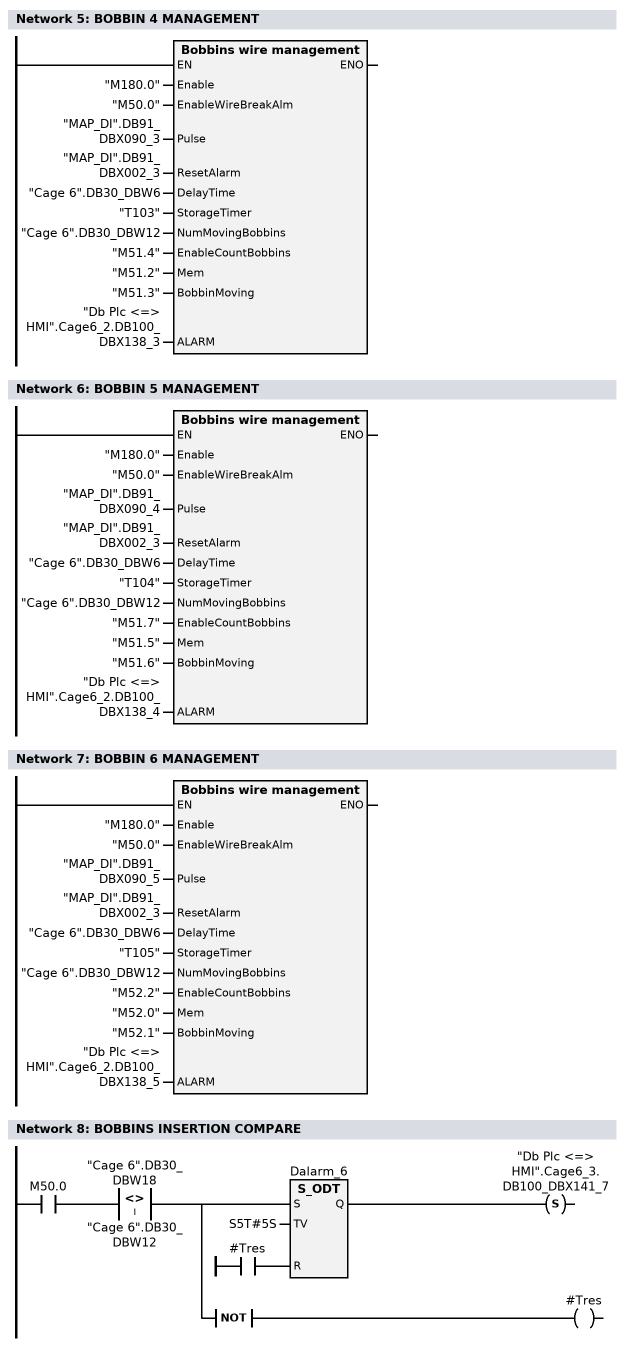
[picture p57: Cage 6 wires insertion networks 5-8]
NETWORK
TITLE = BOBBIN 4 MANAGEMENT
      CALL  "Bobbins wire management" (
           Enable                   := "M180.0",
           EnableWireBreakAlm       := "M50.0",
           Pulse                    := "MAP_DI".DB91_DBX090_3,
           ResetAlarm               := "MAP_DI".DB91_DBX002_3,
           DelayTime                := "Cage 6".DB30_DBW6,
           StorageTimer             := "T103",
           NumMovingBobbins         := "Cage 6".DB30_DBW12,
           EnableCountBobbins       := "M51.4",
           Mem                      := "M51.2",
           BobbinMoving             := "M51.3",
           ALARM                    := "Db Plc <=> HMI".Cage6_2.DB100_DBX138_3);
NETWORK
TITLE = BOBBIN 5 MANAGEMENT
      CALL  "Bobbins wire management" (
           Enable                   := "M180.0",
           EnableWireBreakAlm       := "M50.0",
           Pulse                    := "MAP_DI".DB91_DBX090_4,
           ResetAlarm               := "MAP_DI".DB91_DBX002_3,
           DelayTime                := "Cage 6".DB30_DBW6,
           StorageTimer             := "T104",
           NumMovingBobbins         := "Cage 6".DB30_DBW12,
           EnableCountBobbins       := "M51.7",
           Mem                      := "M51.5",
           BobbinMoving             := "M51.6",
           ALARM                    := "Db Plc <=> HMI".Cage6_2.DB100_DBX138_4);
NETWORK
TITLE = BOBBIN 6 MANAGEMENT
      CALL  "Bobbins wire management" (
           Enable                   := "M180.0",
           EnableWireBreakAlm       := "M50.0",
           Pulse                    := "MAP_DI".DB91_DBX090_5,
           ResetAlarm               := "MAP_DI".DB91_DBX002_3,
           DelayTime                := "Cage 6".DB30_DBW6,
           StorageTimer             := "T105",
           NumMovingBobbins         := "Cage 6".DB30_DBW12,
           EnableCountBobbins       := "M52.2",
           Mem                      := "M52.0",
           BobbinMoving             := "M52.1",
           ALARM                    := "Db Plc <=> HMI".Cage6_2.DB100_DBX138_5);
NETWORK
TITLE = BOBBINS INSERTION COMPARE
      A     "M50.0";
      A(;
      L     "Cage 6".DB30_DBW18;
      L     "Cage 6".DB30_DBW12;
      <>I;
      );
      =     L 1.0;
      A     L 1.0;
      L     S5T#5S;
      SD    "Dalarm_6";
      A     #Tres;
      R     "Dalarm_6";
      NOP   0;
      NOP   0;
      A     "Dalarm_6";
      S     "Db Plc <=> HMI".Cage6_3.DB100_DBX141_7;
      A     L 1.0;
      NOT;
      =     #Tres;
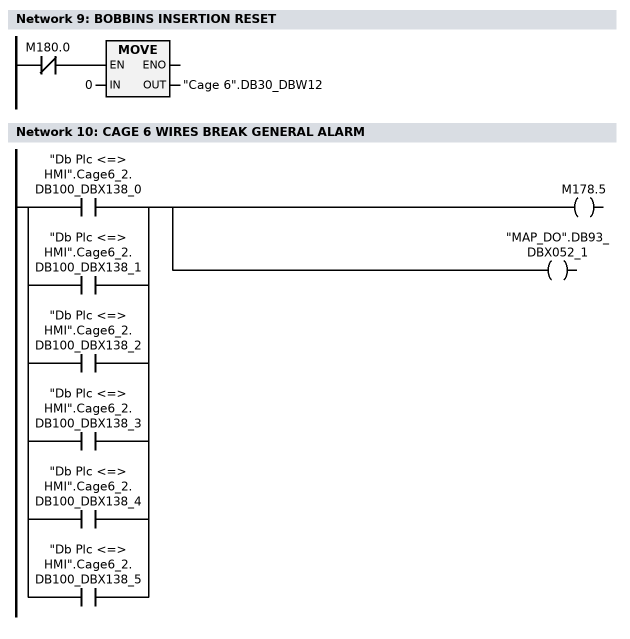
NETWORK
TITLE = BOBBINS INSERTION RESET
      AN    "M180.0";
      JNB   _001;
      L     0;
      T     "Cage 6".DB30_DBW12;
_001: NOP   0;
NETWORK
TITLE = CAGE 6 WIRES BREAK GENERAL ALARM
      O     "Db Plc <=> HMI".Cage6_2.DB100_DBX138_0;
      O     "Db Plc <=> HMI".Cage6_2.DB100_DBX138_1;
      O     "Db Plc <=> HMI".Cage6_2.DB100_DBX138_2;
      O     "Db Plc <=> HMI".Cage6_2.DB100_DBX138_3;
      O     "Db Plc <=> HMI".Cage6_2.DB100_DBX138_4;
      O     "Db Plc <=> HMI".Cage6_2.DB100_DBX138_5;
      =     "M178.5";
      =     "MAP_DO".DB93_DBX052_1;
END_FUNCTION

FUNCTION "Wires break time" : VOID	// FC 74
TITLE = WIRES BREAK TIME FUNCTION
AUTHOR : Milesi
VERSION : 0.1
BEGIN
NETWORK
TITLE = TIME FOR WIRES BREAK CONTROL
//Time for 1 rpm = 60s/Bobbin rpm
//==
//Time for 1 rpm = 60s/(Linear speed/3.141592 * Bobbin Ш)
//==
//Time for 1 rpm = 60/[60000/(3.1415 * 630)] = 1.9792 (s)
//
//In this case for having a good safety margin on the control I do not divide for 
//4 (number fields) but for 3
//
//Time of 1 sector = 1.9792/3 = 0.6597 (s)
//
//Time of 1 sector = K/Linear speed
//==
//K = Linear speed max (mm)*Time of 1 sector (s)/10
//
//K = (60000*0.6597)/10 = 3958.2
//
//Divided 10 for having the time in compatible esadecimale with the base times 
//STEP7 in tenth of second   
      L     3.958200e+03;
      L     "Line".DB55_DBD68;
      /R;
      RND;
      DTB;
      SRW   4;
      L     W#16#1000;
      OW;
      T     "Cage 24".DB15_DBW6;
      T     "Cage 18".DB20_DBW6;
      T     "Cage 12".DB25_DBW6;
      T     "Cage 6".DB30_DBW6;
      T     "Pay-off 630".DB35_DBW6;
END_FUNCTION

FUNCTION "Bobbins diameter" : VOID	// FC 79
TITLE = BOBBINS DIAMETER FUNCTION
AUTHOR : Milesi
VERSION : 0.1
VAR_TEMP
  Enable_24 : BOOL ;
  Enable_18 : BOOL ;
  Enable_12 : BOOL ;
  Enable_6 : BOOL ;
  PayOff_630_Enable : BOOL ;
  PayOff_Enable : BOOL ;
  PayOff_630_Reset : BOOL ;
  PayOff_Reset : BOOL ;
  PayOff_Bobbin_Reset : BOOL ;
END_VAR
BEGIN
NETWORK
TITLE = CAGE 24 DIAMETER CALCULATION
//E47.1 = 4 impulse     
//
      A     "M201.0";
      A     "M192.0";
      =     #Enable_24;
      CALL  "Bobbin diameter calculat" (
           Enable                   := #Enable_24,
           Pulse                    := "MAP_DI".DB91_DBX030_0,
           Pulse_1minute            := "M100.0",
           Reset                    := "M180.7",
           LinearSpeed              := "Line".DB55_DBD68,
           CompattingFactorHMI      := "Cage 24".DB15_DBD28,
           MinDiameterLimit         := 3.550000e+02,
           MaxDiameterLimit         := 6.300000e+02,
           Pulses_number            := 4,
           Mem                      := "M18.4",
           ImpulseForMinRegister    := "Cage 24".DB15_DBW16,
           Diameter                 := "Cage 24".DB15_DBW14);
NETWORK
TITLE = CAGE 18 DIAMETER CALCULATION
//E57.1 = 4 impulse  
      A     "M201.0";
      A     "M186.0";
      =     #Enable_18;
      CALL  "Bobbin diameter calculat" (
           Enable                   := #Enable_18,
           Pulse                    := "MAP_DI".DB91_DBX050_0,
           Pulse_1minute            := "M100.0",
           Reset                    := "M180.6",
           LinearSpeed              := "Line".DB55_DBD68,
           CompattingFactorHMI      := "Cage 18".DB20_DBD28,
           MinDiameterLimit         := 3.550000e+02,
           MaxDiameterLimit         := 6.300000e+02,
           Pulses_number            := 4,
           Mem                      := "M18.3",
           ImpulseForMinRegister    := "Cage 18".DB20_DBW16,
           Diameter                 := "Cage 18".DB20_DBW14);
NETWORK
TITLE = CAGE 12 DIAMETER CALCULATION
//E67.1 = 4 impulse
      A     "M201.0";
      A     "M188.0";
      =     #Enable_12;
      CALL  "Bobbin diameter calculat" (
           Enable                   := #Enable_12,
           Pulse                    := "MAP_DI".DB91_DBX070_0,
           Pulse_1minute            := "M100.0",
           Reset                    := "M180.5",
           LinearSpeed              := "Line".DB55_DBD68,
           CompattingFactorHMI      := "Cage 12".DB25_DBD28,
           MinDiameterLimit         := 3.550000e+02,
           MaxDiameterLimit         := 6.300000e+02,
           Pulses_number            := 4,
           Mem                      := "M18.2",
           ImpulseForMinRegister    := "Cage 12".DB25_DBW16,
           Diameter                 := "Cage 12".DB25_DBW14);
NETWORK
TITLE = CAGE 6 DIAMETER CALCULATION
//E77.1 = 4 impulse 
      A     "M201.0";
      A     "M190.0";
      =     #Enable_6;
      CALL  "Bobbin diameter calculat" (
           Enable                   := #Enable_6,
           Pulse                    := "MAP_DI".DB91_DBX090_0,
           Pulse_1minute            := "M100.0",
           Reset                    := "M180.4",
           LinearSpeed              := "Line".DB55_DBD68,
           CompattingFactorHMI      := 0.000000e+00,
           MinDiameterLimit         := 3.550000e+02,
           MaxDiameterLimit         := 6.300000e+02,
           Pulses_number            := 4,
           Mem                      := "M18.1",
           ImpulseForMinRegister    := "Cage 6".DB30_DBW16,
           Diameter                 := "Cage 6".DB30_DBW14);
NETWORK
TITLE = PAY-OFF 630 DIAMETER CALCULATION
//E79.0 = 4 impulse
      A     "M201.0";
      A     "Pay-off 630".HMI_Bit.DB35_DBX1_7;
      =     #PayOff_630_Enable;
      A     "T0";
      AN    "M180.1";
      AN    "MAP_DI".DB91_DBX099_0;
      =     #PayOff_630_Reset;
      CALL  "Bobbin diameter calculat" (
           Enable                   := #PayOff_630_Enable,
           Pulse                    := "MAP_DI".DB91_DBX099_1,
           Pulse_1minute            := "M100.0",
           Reset                    := #PayOff_630_Reset,
           LinearSpeed              := "Line".DB55_DBD68,
           CompattingFactorHMI      := 0.000000e+00,
           MinDiameterLimit         := 3.550000e+02,
           MaxDiameterLimit         := 6.300000e+02,
           Pulses_number            := 4,
           Mem                      := "M19.0",
           ImpulseForMinRegister    := "Pay-off 630".DB35_DBW16,
           Diameter                 := "Pay-off 630".DB35_DBW14);
NETWORK
TITLE = BOBBINS DIAMETER CALCULATION TIME 
      A     "M201.0";
      AN    "M100.0";
      L     S5T#1M;
      SD    "T5";
      NOP   0;
      NOP   0;
      NOP   0;
      A     "T5";
      =     "M100.0";
END_FUNCTION

FUNCTION "Bobbins brake" : VOID	// FC 80
TITLE = BOBBINS BRAKE OUT FUNCTION
AUTHOR : Milesi
VERSION : 0.1
VAR_TEMP
  Cage12_output : DINT ;
  Cage18_output : DINT ;
  Cage24_output : DINT ;
  pay_of_630_output : DINT ;
  Cage6_output : DINT ;
  pay_bobbin_output : DINT ;
END_VAR
BEGIN
NETWORK
TITLE = CAGE 24 BOBBINS BRAKES OUTPUT
      L     "Cage 24".DB15_DBD128;
      L     "Cage 24".DB15_DBW14;
      ITD;
      DTR;
      *R;
      L     6.300000e+04;
      /R;
      L     2.764800e+04;
      *R;
      RND;
      L     27648;
      >=D;
      JC    OUT1;
      TAK;
OUT1: T     "-659Y2";
NETWORK
TITLE = CAGE 18 BOBBINS BRAKES OUTPUT
      L     "Cage 18".DB20_DBD128;
      L     "Cage 18".DB20_DBW14;
      ITD;
      DTR;
      *R;
      L     6.300000e+04;
      /R;
      L     2.764800e+04;
      *R;
      RND;
      L     27648;
      >=D;
      JC    OUT2;
      TAK;
OUT2: T     "-559Y2";
NETWORK
TITLE = CAGE 12 BOBBINS BRAKES OUTPUT
      L     "Cage 12".DB25_DBD128;
      L     "Cage 12".DB25_DBW14;
      ITD;
      DTR;
      *R;
      L     6.300000e+04;
      /R;
      L     2.764800e+04;
      *R;
      RND;
      L     27648;
      >=D;
      JC    OUT3;
      TAK;
OUT3: T     "PAW288";
NETWORK
TITLE = CAGE 6 BOBBINS BRAKES OUTPUT
      L     "Cage 6".DB30_DBD128;
      L     "Cage 6".DB30_DBW14;
      ITD;
      DTR;
      *R;
      L     6.300000e+04;
      /R;
      L     2.764800e+04;
      *R;
      RND;
      L     27648;
      >=D;
      JC    OUT4;
      TAK;
OUT4: T     "-359Y2";
NETWORK
TITLE = PAY-OFF 630 BOBBIN BRAKE OUTPUT
      L     "Pay-off 630".DB35_DBD20;
      L     "Pay-off 630".DB35_DBW14;
      ITD;
      DTR;
      *R;
      L     6.300000e+04;
      /R;
      L     2.764800e+04;
      *R;
      RND;
      L     27648;
      >=D;
      JC    OUT5;
      TAK;
OUT5: AN    "MAP_DI".DB91_DBX099_4;
      O     "M180.1";
      JC    OUT6;
      L     0;
OUT6: T     "-359Y4";
END_FUNCTION

FUNCTION "Rpm increase" : VOID	// FC 81
TITLE = RPM INCREASE FUNCTION
AUTHOR : Milesi
VERSION : 0.1
VAR_TEMP
  Time_sec : INT ;	//Minuts in seconds
END_VAR
BEGIN
NETWORK
TITLE = STEP TO MAKE 
//Bobbin max Ш - Bobbin min Ш
//630 - 355 = 275
      L     2.750000e+02;
      L     "Line".DB55_DBD156;
      /R;
      T     "Line".DB55_DBD176;
      L     1.000000e+00;
      -R;
      T     "Line".DB55_DBD184;
NETWORK
TITLE = LINEAR SPEED INCREASE FOR SINGLE STEP 
      L     "Line".DB55_DBD40;
      L     "Line".DB55_DBD72;
      -R;
      L     "Line".DB55_DBD184;
      /R;
      T     "Line".DB55_DBD196;
NETWORK
TITLE = LINEAR SPEED INCREASE CONTROL TIME
      A     "M180.1";
      A     "M201.0";
      JNB   OUT;
      A     "M3.5";
      JNB   CLOC;
      L     "Line".DB55_DBD168;
      L     1.000000e+00;
      +R;
      T     "Line".DB55_DBD168;
CLOC: JU    EXIT;
NETWORK
TITLE = LINEAR SPEED INCREASE PARAMETERS RESET
OUT:  L     0.000000e+00;
      T     "Line".DB55_DBD168;
      A     "M180.1";
      JC    EXIT;
      L     6.300000e+02;
      T     "Line".DB55_DBD172;
      L     0.000000e+00;
      T     "Line".DB55_DBD164;
      L     0.000000e+00;
      T     "Line".DB55_DBD76;
EXIT: NOP   0;
NETWORK
TITLE = LINEAR SPEED INCREASE TIME MINUTS TO SECONDS COVERSION
      L     "Line".DB55_DBD160;
      RND;
      T     #Time_sec;
NETWORK
TITLE = DIAMETER NEXT STEP
      L     "Line".DB55_DBD172;
      L     "Line".DB55_DBD156;
      -R;
      T     "Line".DB55_DBD188;
NETWORK
TITLE = LINEAR SPEED INCREASE CONTROL 
      L     "Line".DB55_DBD168;
      RND;
      L     #Time_sec;
      <I;
      BEC;
      L     0.000000e+00;
      T     "Line".DB55_DBD168;
NETWORK
TITLE = LINE LINEAR SPEED INCREASE
      A(;
      L     "Line".DB55_DBD188;
      L     "Line".DB55_DBD192;
      <R;
      );
      O(;
      L     "Line".DB55_DBD164;
      L     "Line".DB55_DBD184;
      >=R;
      );
      BEC;
      L     "Line".DB55_DBD164;
      L     1.000000e+00;
      +R;
      T     "Line".DB55_DBD164;
      L     "Line".DB55_DBD188;
      T     "Line".DB55_DBD172;
      L     "Line".DB55_DBD164;
      L     "Line".DB55_DBD196;
      *R;
      T     "Line".DB55_DBD76;
END_FUNCTION

FUNCTION "Map Input Function" : VOID	// FC 91
TITLE = MAP INPUT FUNCTION
VERSION : 0.1
VAR_TEMP
  Temp1 : BOOL ;
END_VAR
BEGIN
NETWORK
TITLE = da DB91.dbx0.0 a DB91.dbx0.7
      A     "-126K1:Auxiliary";
      =     "MAP_DI".DB91_DBX000_0;
      A     "-126K4";
      =     "MAP_DI".DB91_DBX000_1;
      A     "-175S3";
      =     "MAP_DI".DB91_DBX000_2;
      A     "-112Q3";
      =     "MAP_DI".DB91_DBX000_3;
      A     "-108G1:Alarm";
      =     "MAP_DI".DB91_DBX000_4;
      A     "-108G1:Bat ok";
      =     "MAP_DI".DB91_DBX000_5;
      A     "-116Q1";
      =     "MAP_DI".DB91_DBX000_6;
      CLR;
      =     "MAP_DI".DB91_DBX000_7;
NETWORK
TITLE = da DB91.dbx1.0 a DB91.dbx1.7
      A     "-119Q1";
      =     "MAP_DI".DB91_DBX001_0;
      A     "-141R1:T2";
      =     "MAP_DI".DB91_DBX001_1;
      A     "-140G1:X104:20";
      =     "MAP_DI".DB91_DBX001_2;
      CLR;
      =     "MAP_DI".DB91_DBX001_3;
      =     "MAP_DI".DB91_DBX001_4;
      =     "MAP_DI".DB91_DBX001_5;
      =     "MAP_DI".DB91_DBX001_6;
      =     "MAP_DI".DB91_DBX001_7;
NETWORK
TITLE = da DB91.dbx2.0 a DB91.dbx2.7
      A     "-177S1";
      =     "MAP_DI".DB91_DBX002_0;
      A     "-177S2";
      =     "MAP_DI".DB91_DBX002_1;
      A     "-177S3";
      =     "MAP_DI".DB91_DBX002_2;
      A     "-177S4";
      =     "MAP_DI".DB91_DBX002_3;
      A     "-177S5";
      =     "MAP_DI".DB91_DBX002_4;
      A     "-112K1";
      =     "MAP_DI".DB91_DBX002_5;
      A     "-112K1:66";
      =     "MAP_DI".DB91_DBX002_6;
      A     "-113G1:4";
      =     "MAP_DI".DB91_DBX002_7;
NETWORK
TITLE = da DB91.dbx3.0 a DB91.dbx3.7
      A     "-113G1:3";
      =     "MAP_DI".DB91_DBX003_0;
      A     "-109Q6";
      =     "MAP_DI".DB91_DBX003_1;
      A     "-115Q1";
      =     "MAP_DI".DB91_DBX003_2;
      A     "-140Q1";
      =     "MAP_DI".DB91_DBX003_3;
      A     "-109Q2";
      =     "MAP_DI".DB91_DBX003_4;
      CLR;
      =     "MAP_DI".DB91_DBX003_5;
      =     "MAP_DI".DB91_DBX003_6;
      =     "MAP_DI".DB91_DBX003_7;
NETWORK
TITLE = da DB91.dbx4.0 a DB91.dbx4.7
      A     "-922S5";
      =     "MAP_DI".DB91_DBX004_0;
      A     "-922S6";
      =     "MAP_DI".DB91_DBX004_1;
      A     "-922S7";
      =     "MAP_DI".DB91_DBX004_2;
      A     "-922S8";
      =     "MAP_DI".DB91_DBX004_3;
      A     "-945Q1";
      =     "MAP_DI".DB91_DBX004_4;
      A     "-941Q2";
      =     "MAP_DI".DB91_DBX004_5;
      A     "-964S1:Forward";
      =     "MAP_DI".DB91_DBX004_6;
      A     "-964S1:Backward";
      =     "MAP_DI".DB91_DBX004_7;
NETWORK
TITLE = da DB91.dbx5.0 a DB91.dbx5.7
      L     B#16#0;
      T     DB91.DBB 5;
NETWORK
TITLE = da DB91.dbx6.0 a DB91.dbx6.7
      A     "-961S1";
      =     "MAP_DI".DB91_DBX006_0;
      A     "-961S2";
      =     "MAP_DI".DB91_DBX006_1;
      A     "-961S3";
      =     "MAP_DI".DB91_DBX006_2;
      A     "-961S4";
      =     "MAP_DI".DB91_DBX006_3;
      A     "-961S5:UP";
      =     "MAP_DI".DB91_DBX006_4;
      A     "-961S5:DOWN";
      =     "MAP_DI".DB91_DBX006_5;
      A     "-961S7:UP";
      =     "MAP_DI".DB91_DBX006_6;
      A     "-961S7:DOWN";
      =     "MAP_DI".DB91_DBX006_7;
NETWORK
TITLE = da DB91.dbx7.0 a DB91.dbx7.7
      A     "-962S1:UP";
      =     "MAP_DI".DB91_DBX007_0;
      A     "-962S1:DOWN";
      =     "MAP_DI".DB91_DBX007_1;
      A     "-962S3:OPEN";
      =     "MAP_DI".DB91_DBX007_2;
      A     "-962S3:CLOSE";
      =     "MAP_DI".DB91_DBX007_3;
      A     "-962S5";
      =     "MAP_DI".DB91_DBX007_4;
      A     "-962S6";
      =     "MAP_DI".DB91_DBX007_5;
      CLR;
      =     "MAP_DI".DB91_DBX007_6;
      =     "MAP_DI".DB91_DBX007_7;
NETWORK
TITLE = da DB91.dbx8.0 a DB91.dbx8.7
      A     "-962S7";
      =     "MAP_DI".DB91_DBX008_0;
      A     "-962S8";
      =     "MAP_DI".DB91_DBX008_1;
      A     "-922S3";
      =     "MAP_DI".DB91_DBX008_2;
      A     "-922S4";
      =     "MAP_DI".DB91_DBX008_3;
      A     "-964B3";
      =     "MAP_DI".DB91_DBX008_4;
      A     "-964B4";
      =     "MAP_DI".DB91_DBX008_5;
      A     "-945Q2";
      =     "MAP_DI".DB91_DBX008_6;
      CLR;
      =     "MAP_DI".DB91_DBX008_7;
NETWORK
TITLE = da DB91.dbx9.0 a DB91.dbx9.7
      CLR;
      =     "MAP_DI".DB91_DBX009_0;
      A     "-944Q1";
      =     "MAP_DI".DB91_DBX009_1;
      A     "-112Q8";
      =     "MAP_DI".DB91_DBX009_2;
      A     "-109Q7";
      =     "MAP_DI".DB91_DBX009_3;
      CLR;
      =     "MAP_DI".DB91_DBX009_4;
      =     "MAP_DI".DB91_DBX009_5;
      =     "MAP_DI".DB91_DBX009_6;
      =     "MAP_DI".DB91_DBX009_7;
NETWORK
TITLE = da DB91.dbx10.0 a DB91.dbx10.7
      L     B#16#0;
      T     DB91.DBB 10;
NETWORK
TITLE = da DB91.dbx11.0 a DB91.dbx11.7
      L     B#16#0;
      T     DB91.DBB 11;
NETWORK
TITLE = da DB91.dbx12.0 a DB91.dbx12.7
      A     "-705Q1";
      =     "MAP_DI".DB91_DBX012_0;
      A     "-718S4";
      =     "MAP_DI".DB91_DBX012_1;
      A     "-718S5";
      =     "MAP_DI".DB91_DBX012_2;
      A     "-718B6";
      =     "MAP_DI".DB91_DBX012_3;
      A     "-177S6";
      =     "MAP_DI".DB91_DBX012_4;
      A     "-177S7:Forward";
      =     "MAP_DI".DB91_DBX012_5;
      A     "-177S7:Backward";
      =     "MAP_DI".DB91_DBX012_6;
      CLR;
      =     "MAP_DI".DB91_DBX012_7;
NETWORK
TITLE = da DB91.dbx13.0 a DB91.dbx13.7
      L     B#16#0;
      T     DB91.DBB 13;
NETWORK
TITLE = da DB91.dbx14.0 a DB91.dbx14.7
      L     B#16#0;
      T     DB91.DBB 14;
NETWORK
TITLE = da DB91.dbx15.0 a DB91.dbx15.7
      L     B#16#0;
      T     DB91.DBB 15;
NETWORK
TITLE = da DB91.dbx16.0 a DB91.dbx16.7
      L     B#16#0;
      T     DB91.DBB 16;
NETWORK
TITLE = da DB91.dbx17.0 a DB91.dbx17.7
      L     B#16#0;
      T     DB91.DBB 17;
NETWORK
TITLE = da DB91.dbx18.0 a DB91.dbx18.7
      A     "-640Q1";
      =     "MAP_DI".DB91_DBX018_0;
      A     "-109Q12";
      =     "MAP_DI".DB91_DBX018_1;
      A     "-605Q2";
      =     "MAP_DI".DB91_DBX018_2;
      A     "-605Q1";
      =     "MAP_DI".DB91_DBX018_3;
      A     "-607Q2";
      =     "MAP_DI".DB91_DBX018_4;
      A     "-607Q1";
      =     "MAP_DI".DB91_DBX018_5;
      CLR;
      =     "MAP_DI".DB91_DBX018_6;
      A     "-606Q1";
      =     "MAP_DI".DB91_DBX018_7;
NETWORK
TITLE = da DB91.dbx19.0 a DB91.dbx19.7
      L     B#16#0;
      T     DB91.DBB 19;
NETWORK
TITLE = da DB91.dbx20.0 a DB91.dbx20.7
      A     "-661S1";
      =     "MAP_DI".DB91_DBX020_0;
      A     "-661S2";
      =     "MAP_DI".DB91_DBX020_1;
      A     "-661S3";
      =     "MAP_DI".DB91_DBX020_2;
      A     "-661S4";
      =     "MAP_DI".DB91_DBX020_3;
      A     "-661S5";
      =     "MAP_DI".DB91_DBX020_4;
      A     "-661S6";
      =     "MAP_DI".DB91_DBX020_5;
      A     "-661S7";
      =     "MAP_DI".DB91_DBX020_6;
      A     "-661S8";
      =     "MAP_DI".DB91_DBX020_7;
NETWORK
TITLE = da DB91.dbx21.0 a DB91.dbx21.7
      A     "-662B1";
      =     "MAP_DI".DB91_DBX021_0;
      A     "-662B2";
      =     "MAP_DI".DB91_DBX021_1;
      A     "-662S3";
      =     "MAP_DI".DB91_DBX021_2;
      A     "-686Y1";
      =     "MAP_DI".DB91_DBX021_3;
      A     "-662S5";
      =     "MAP_DI".DB91_DBX021_4;
      A     "-662S6";
      =     "MAP_DI".DB91_DBX021_5;
      A     "-662B7";
      =     "MAP_DI".DB91_DBX021_6;
      A     "-662B8";
      =     "MAP_DI".DB91_DBX021_7;
NETWORK
TITLE = da DB91.dbx22.0 a DB91.dbx22.7
      A     "-663S1";
      =     "MAP_DI".DB91_DBX022_0;
      A     "-663S2";
      =     "MAP_DI".DB91_DBX022_1;
      A     "-663S3";
      =     "MAP_DI".DB91_DBX022_2;
      A     "-663S4";
      =     "MAP_DI".DB91_DBX022_3;
      A     "-663S5:CLOSING";
      =     "MAP_DI".DB91_DBX022_4;
      A     "-663S5:OPENING";
      =     "MAP_DI".DB91_DBX022_5;
      A     "-663S7:CLOSING";
      =     "MAP_DI".DB91_DBX022_6;
      A     "-663S7:OPENING";
      =     "MAP_DI".DB91_DBX022_7;
NETWORK
TITLE = da DB91.dbx23.0 a DB91.dbx23.7
      A     "-664S1:CLOSING";
      =     "MAP_DI".DB91_DBX023_0;
      A     "-664S1:OPENING";
      =     "MAP_DI".DB91_DBX023_1;
      CLR;
      =     "MAP_DI".DB91_DBX023_2;
      =     "MAP_DI".DB91_DBX023_3;
      =     "MAP_DI".DB91_DBX023_4;
      =     "MAP_DI".DB91_DBX023_5;
      A     "-664S7";
      =     "MAP_DI".DB91_DBX023_6;
      CLR;
      =     "MAP_DI".DB91_DBX023_7;
NETWORK
TITLE = da DB91.dbx24.0 a DB91.dbx24.7
      CLR;
      =     "MAP_DI".DB91_DBX024_0;
      =     "MAP_DI".DB91_DBX024_1;
      =     "MAP_DI".DB91_DBX024_2;
      =     "MAP_DI".DB91_DBX024_3;
      =     "MAP_DI".DB91_DBX024_4;
      =     "MAP_DI".DB91_DBX024_5;
      A     "-688Y8";
      =     "MAP_DI".DB91_DBX024_6;
      A     "-665S8";
      =     "MAP_DI".DB91_DBX024_7;
NETWORK
TITLE = da DB91.dbx25.0 a DB91.dbx25.7
      A     "-666S1";
      =     "MAP_DI".DB91_DBX025_0;
      A     "-666S2";
      =     "MAP_DI".DB91_DBX025_1;
      CLR;
      =     "MAP_DI".DB91_DBX025_2;
      =     "MAP_DI".DB91_DBX025_3;
      =     "MAP_DI".DB91_DBX025_4;
      =     "MAP_DI".DB91_DBX025_5;
      =     "MAP_DI".DB91_DBX025_6;
      =     "MAP_DI".DB91_DBX025_7;
NETWORK
TITLE = da DB91.dbx26.0 a DB91.dbx26.7
      L     B#16#0;
      T     DB91.DBB 26;
NETWORK
TITLE = da DB91.dbx27.0 a DB91.dbx27.7
      CLR;
      =     "MAP_DI".DB91_DBX027_0;
      =     "MAP_DI".DB91_DBX027_1;
      =     "MAP_DI".DB91_DBX027_2;
      =     "MAP_DI".DB91_DBX027_3;
      A     "-670S1";
      =     "MAP_DI".DB91_DBX027_4;
      A     "-670S2";
      =     "MAP_DI".DB91_DBX027_5;
      A     "-670S3";
      =     "MAP_DI".DB91_DBX027_6;
      A     "-670S4";
      =     "MAP_DI".DB91_DBX027_7;
NETWORK
TITLE = da DB91.dbx28.0 a DB91.dbx28.7
      L     B#16#0;
      T     DB91.DBB 28;
NETWORK
TITLE = da DB91.dbx29.0 a DB91.dbx29.7
      L     B#16#0;
      T     DB91.DBB 29;
NETWORK
TITLE = da DB91.dbx30.0 a DB91.dbx30.7
      A     "-667B1";
      =     "MAP_DI".DB91_DBX030_0;
      A     "-667B2";
      =     "MAP_DI".DB91_DBX030_1;
      A     "-667B3";
      =     "MAP_DI".DB91_DBX030_2;
      A     "-667B4";
      =     "MAP_DI".DB91_DBX030_3;
      A     "-667B5";
      =     "MAP_DI".DB91_DBX030_4;
      A     "-667B6";
      =     "MAP_DI".DB91_DBX030_5;
      A     "-667B7";
      =     "MAP_DI".DB91_DBX030_6;
      A     "-667B8";
      =     "MAP_DI".DB91_DBX030_7;
NETWORK
TITLE = da DB91.dbx31.0 a DB91.dbx31.7
      A     "-668B1";
      =     "MAP_DI".DB91_DBX031_0;
      A     "-668B2";
      =     "MAP_DI".DB91_DBX031_1;
      A     "-668B3";
      =     "MAP_DI".DB91_DBX031_2;
      A     "-668B4";
      =     "MAP_DI".DB91_DBX031_3;
      A     "-668B5";
      =     "MAP_DI".DB91_DBX031_4;
      A     "-668B6";
      =     "MAP_DI".DB91_DBX031_5;
      A     "-668B7";
      =     "MAP_DI".DB91_DBX031_6;
      A     "-668B8";
      =     "MAP_DI".DB91_DBX031_7;
NETWORK
TITLE = da DB91.dbx32.0 a DB91.dbx32.7
      A     "-669B1";
      =     "MAP_DI".DB91_DBX032_0;
      A     "-669B2";
      =     "MAP_DI".DB91_DBX032_1;
      A     "-669B3";
      =     "MAP_DI".DB91_DBX032_2;
      A     "-669B4";
      =     "MAP_DI".DB91_DBX032_3;
      A     "-669B5";
      =     "MAP_DI".DB91_DBX032_4;
      A     "-669B6";
      =     "MAP_DI".DB91_DBX032_5;
      A     "-669B7";
      =     "MAP_DI".DB91_DBX032_6;
      A     "-669B8";
      =     "MAP_DI".DB91_DBX032_7;
NETWORK
TITLE = da DB91.dbx33.0 a DB91.dbx33.7
      L     B#16#0;
      T     DB91.DBB 33;
NETWORK
TITLE = da DB91.dbx34.0 a DB91.dbx34.7
      L     B#16#0;
      T     DB91.DBB 34;
NETWORK
TITLE = da DB91.dbx35.0 a DB91.dbx35.7
      L     B#16#0;
      T     DB91.DBB 35;
NETWORK
TITLE = da DB91.dbx36.0 a DB91.dbx36.7
      A     "+MCB24:7";
      =     "MAP_DI".DB91_DBX036_0;
      A     "+MCB24:8";
      =     "MAP_DI".DB91_DBX036_1;
      A     "+MCB24:9";
      =     "MAP_DI".DB91_DBX036_2;
      A     "+MCB24:10";
      =     "MAP_DI".DB91_DBX036_3;
      CLR;
      =     "MAP_DI".DB91_DBX036_4;
      =     "MAP_DI".DB91_DBX036_5;
      =     "MAP_DI".DB91_DBX036_6;
      =     "MAP_DI".DB91_DBX036_7;
NETWORK
TITLE = da DB91.dbx37.0 a DB91.dbx37.7
      L     B#16#0;
      T     DB91.DBB 37;
NETWORK
TITLE = da DB91.dbx38.0 a DB91.dbx38.7
      A     "-540Q1";
      =     "MAP_DI".DB91_DBX038_0;
      A     "-109Q11";
      =     "MAP_DI".DB91_DBX038_1;
      A     "-505Q2";
      =     "MAP_DI".DB91_DBX038_2;
      A     "-505Q1";
      =     "MAP_DI".DB91_DBX038_3;
      A     "-507Q2";
      =     "MAP_DI".DB91_DBX038_4;
      A     "-507Q1";
      =     "MAP_DI".DB91_DBX038_5;
      CLR;
      =     "MAP_DI".DB91_DBX038_6;
      A     "-506Q1";
      =     "MAP_DI".DB91_DBX038_7;
NETWORK
TITLE = da DB91.dbx39.0 a DB91.dbx39.7
      L     B#16#0;
      T     DB91.DBB 39;
NETWORK
TITLE = da DB91.dbx40.0 a DB91.dbx40.7
      A     "-561S1";
      =     "MAP_DI".DB91_DBX040_0;
      A     "-561S2";
      =     "MAP_DI".DB91_DBX040_1;
      A     "-561S3";
      =     "MAP_DI".DB91_DBX040_2;
      A     "-561S4";
      =     "MAP_DI".DB91_DBX040_3;
      A     "-561S5";
      =     "MAP_DI".DB91_DBX040_4;
      A     "-561B6";
      =     "MAP_DI".DB91_DBX040_5;
      A     "-561B7";
      =     "MAP_DI".DB91_DBX040_6;
      A     "-561S8";
      =     "MAP_DI".DB91_DBX040_7;
NETWORK
TITLE = da DB91.dbx41.0 a DB91.dbx41.7
      A     "-562B1";
      =     "MAP_DI".DB91_DBX041_0;
      A     "-562B2";
      =     "MAP_DI".DB91_DBX041_1;
      A     "-562S3";
      =     "MAP_DI".DB91_DBX041_2;
      A     "-586Y1";
      =     "MAP_DI".DB91_DBX041_3;
      A     "-562S5";
      =     "MAP_DI".DB91_DBX041_4;
      A     "-562S6";
      =     "MAP_DI".DB91_DBX041_5;
      A     "-562B7";
      =     "MAP_DI".DB91_DBX041_6;
      A     "-562B8";
      =     "MAP_DI".DB91_DBX041_7;
NETWORK
TITLE = da DB91.dbx42.0 a DB91.dbx42.7
      A     "-563S1";
      =     "MAP_DI".DB91_DBX042_0;
      A     "-563S2";
      =     "MAP_DI".DB91_DBX042_1;
      A     "-563S3";
      =     "MAP_DI".DB91_DBX042_2;
      A     "-563S4";
      =     "MAP_DI".DB91_DBX042_3;
      A     "-563S5:CLOSING";
      =     "MAP_DI".DB91_DBX042_4;
      A     "-563S5:OPENING";
      =     "MAP_DI".DB91_DBX042_5;
      A     "-563S7:CLOSING";
      =     "MAP_DI".DB91_DBX042_6;
      A     "-563S7:OPENING";
      =     "MAP_DI".DB91_DBX042_7;
NETWORK
TITLE = da DB91.dbx43.0 a DB91.dbx43.7
      A     "-564S1:CLOSING";
      =     "MAP_DI".DB91_DBX043_0;
      A     "-563S1:OPENING";
      =     "MAP_DI".DB91_DBX043_1;
      CLR;
      =     "MAP_DI".DB91_DBX043_2;
      CLR;
      =     "MAP_DI".DB91_DBX043_3;
      CLR;
      =     "MAP_DI".DB91_DBX043_4;
      CLR;
      =     "MAP_DI".DB91_DBX043_5;
      A     "-564S7";
      =     "MAP_DI".DB91_DBX043_6;
      CLR;
      =     "MAP_DI".DB91_DBX043_7;
NETWORK
TITLE = da DB91.dbx44.0 a DB91.dbx44.7
      CLR;
      =     "MAP_DI".DB91_DBX044_0;
      =     "MAP_DI".DB91_DBX044_1;
      =     "MAP_DI".DB91_DBX044_2;
      =     "MAP_DI".DB91_DBX044_3;
      =     "MAP_DI".DB91_DBX044_4;
      =     "MAP_DI".DB91_DBX044_5;
      A     "-588Y8";
      =     "MAP_DI".DB91_DBX044_6;
      A     "-565S8";
      =     "MAP_DI".DB91_DBX044_7;
NETWORK
TITLE = da DB91.dbx45.0 a DB91.dbx45.7
      A     "-566S1";
      =     "MAP_DI".DB91_DBX045_0;
      A     "-566S2";
      =     "MAP_DI".DB91_DBX045_1;
      CLR;
      =     "MAP_DI".DB91_DBX045_2;
      =     "MAP_DI".DB91_DBX045_3;
      =     "MAP_DI".DB91_DBX045_4;
      =     "MAP_DI".DB91_DBX045_5;
      =     "MAP_DI".DB91_DBX045_6;
      =     "MAP_DI".DB91_DBX045_7;
NETWORK
TITLE = da DB91.dbx46.0 a DB91.dbx46.7
      L     B#16#0;
      T     DB91.DBB 46;
NETWORK
TITLE = da DB91.dbx47.0 a DB91.dbx47.7
      A     "-569S3";
      =     "MAP_DI".DB91_DBX047_0;
      A     "-569S4";
      =     "MAP_DI".DB91_DBX047_1;
      A     "-569S5";
      =     "MAP_DI".DB91_DBX047_2;
      A     "-569S6";
      =     "MAP_DI".DB91_DBX047_3;
      CLR;
      =     "MAP_DI".DB91_DBX047_4;
      =     "MAP_DI".DB91_DBX047_5;
      =     "MAP_DI".DB91_DBX047_6;
      =     "MAP_DI".DB91_DBX047_7;
NETWORK
TITLE = da DB91.dbx48.0 a DB91.dbx48.7
      L     B#16#0;
      T     DB91.DBB 48;
NETWORK
TITLE = da DB91.dbx49.0 a DB91.dbx49.7
      L     B#16#0;
      T     DB91.DBB 49;
NETWORK
TITLE = da DB91.dbx50.0 a DB91.dbx50.7
      A     "-567B1";
      =     "MAP_DI".DB91_DBX050_0;
      A     "-567B2";
      =     "MAP_DI".DB91_DBX050_1;
      A     "-567B3";
      =     "MAP_DI".DB91_DBX050_2;
      A     "-567B4";
      =     "MAP_DI".DB91_DBX050_3;
      A     "-567B5";
      =     "MAP_DI".DB91_DBX050_4;
      A     "-567B6";
      =     "MAP_DI".DB91_DBX050_5;
      A     "-567B7";
      =     "MAP_DI".DB91_DBX050_6;
      A     "-567B8";
      =     "MAP_DI".DB91_DBX050_7;
NETWORK
TITLE = da DB91.dbx51.0 a DB91.dbx51.7
      A     "-568B1";
      =     "MAP_DI".DB91_DBX051_0;
      A     "-568B2";
      =     "MAP_DI".DB91_DBX051_1;
      A     "-568B3";
      =     "MAP_DI".DB91_DBX051_2;
      A     "-568B4";
      =     "MAP_DI".DB91_DBX051_3;
      A     "-568B5";
      =     "MAP_DI".DB91_DBX051_4;
      A     "-568B6";
      =     "MAP_DI".DB91_DBX051_5;
      A     "-568B7";
      =     "MAP_DI".DB91_DBX051_6;
      A     "-568B8";
      =     "MAP_DI".DB91_DBX051_7;
NETWORK
TITLE = da DB91.dbx52.0 a DB91.dbx52.7
      A     "-569B1";
      =     "MAP_DI".DB91_DBX052_0;
      A     "-569B2";
      =     "MAP_DI".DB91_DBX052_1;
      CLR;
      =     "MAP_DI".DB91_DBX052_2;
      CLR;
      =     "MAP_DI".DB91_DBX052_3;
      CLR;
      =     "MAP_DI".DB91_DBX052_4;
      CLR;
      =     "MAP_DI".DB91_DBX052_5;
      CLR;
      =     "MAP_DI".DB91_DBX052_6;
      CLR;
      =     "MAP_DI".DB91_DBX052_7;
NETWORK
TITLE = da DB91.dbx53.0 a DB91.dbx53.7
      L     B#16#0;
      T     DB91.DBB 53;
NETWORK
TITLE = da DB91.dbx54.0 a DB91.dbx54.7
      L     B#16#0;
      T     DB91.DBB 54;
NETWORK
TITLE = da DB91.dbx55.0 a DB91.dbx55.7
      L     B#16#0;
      T     DB91.DBB 55;
NETWORK
TITLE = da DB91.dbx56.0 a DB91.dbx56.7
      A     "+MCB18:7";
      =     "MAP_DI".DB91_DBX056_0;
      A     "+MCB18:8";
      =     "MAP_DI".DB91_DBX056_1;
      A     "+MCB18:9";
      =     "MAP_DI".DB91_DBX056_2;
      A     "+MCB18:10";
      =     "MAP_DI".DB91_DBX056_3;
      A     "-565B5";
      =     "MAP_DI".DB91_DBX056_4;
      A     "-565B6";
      =     "MAP_DI".DB91_DBX056_5;
      CLR;
      =     "MAP_DI".DB91_DBX056_6;
      CLR;
      =     "MAP_DI".DB91_DBX056_7;
NETWORK
TITLE = da DB91.dbx57.0 a DB91.dbx57.7
      L     B#16#0;
      T     DB91.DBB 57;
NETWORK
TITLE = da DB91.dbx58.0 a DB91.dbx58.7
      A     "-440Q1";
      =     "MAP_DI".DB91_DBX058_0;
      A     "-109Q10";
      =     "MAP_DI".DB91_DBX058_1;
      A     "-405Q2";
      =     "MAP_DI".DB91_DBX058_2;
      A     "-405Q1";
      =     "MAP_DI".DB91_DBX058_3;
      A     "-407Q2";
      =     "MAP_DI".DB91_DBX058_4;
      A     "-407Q1";
      =     "MAP_DI".DB91_DBX058_5;
      CLR;
      =     "MAP_DI".DB91_DBX058_6;
      A     "-406Q1";
      =     "MAP_DI".DB91_DBX058_7;
NETWORK
TITLE = da DB91.dbx59.0 a DB91.dbx59.7
      L     B#16#0;
      T     DB91.DBB 59;
NETWORK
TITLE = da DB91.dbx60.0 a DB91.dbx60.7
      A     "-461S1";
      =     "MAP_DI".DB91_DBX060_0;
      A     "-461S2";
      =     "MAP_DI".DB91_DBX060_1;
      A     "-461S3";
      =     "MAP_DI".DB91_DBX060_2;
      A     "-461S4";
      =     "MAP_DI".DB91_DBX060_3;
      A     "-461S5";
      =     "MAP_DI".DB91_DBX060_4;
      A     "-461B6";
      =     "MAP_DI".DB91_DBX060_5;
      A     "-461B7";
      =     "MAP_DI".DB91_DBX060_6;
      A     "-461S8";
      =     "MAP_DI".DB91_DBX060_7;
NETWORK
TITLE = da DB91.dbx61.0 a DB91.dbx61.7
      A     "-462B1";
      =     "MAP_DI".DB91_DBX061_0;
      A     "-462B2";
      =     "MAP_DI".DB91_DBX061_1;
      A     "-462S3";
      =     "MAP_DI".DB91_DBX061_2;
      A     "-486Y1";
      =     "MAP_DI".DB91_DBX061_3;
      A     "-462S5";
      =     "MAP_DI".DB91_DBX061_4;
      A     "-462S6";
      =     "MAP_DI".DB91_DBX061_5;
      A     "-462B7";
      =     "MAP_DI".DB91_DBX061_6;
      A     "-462B8";
      =     "MAP_DI".DB91_DBX061_7;
NETWORK
TITLE = da DB91.dbx62.0 a DB91.dbx62.7
      A     "-463S1";
      =     "MAP_DI".DB91_DBX062_0;
      A     "-463S2";
      =     "MAP_DI".DB91_DBX062_1;
      A     "-463S3";
      =     "MAP_DI".DB91_DBX062_2;
      A     "-463S4";
      =     "MAP_DI".DB91_DBX062_3;
      A     "-463S5:CLOSING";
      =     "MAP_DI".DB91_DBX062_4;
      A     "-463S5:OPENING";
      =     "MAP_DI".DB91_DBX062_5;
      A     "-463S7:CLOSING";
      =     "MAP_DI".DB91_DBX062_6;
      A     "-463S7:OPENING";
      =     "MAP_DI".DB91_DBX062_7;
NETWORK
TITLE = da DB91.dbx63.0 a DB91.dbx63.7
      A     "-464S1:CLOSING";
      =     "MAP_DI".DB91_DBX063_0;
      A     "-464S1:OPENING";
      =     "MAP_DI".DB91_DBX063_1;
      CLR;
      =     "MAP_DI".DB91_DBX063_2;
      =     "MAP_DI".DB91_DBX063_3;
      =     "MAP_DI".DB91_DBX063_4;
      =     "MAP_DI".DB91_DBX063_5;
      A     "-464S7";
      =     "MAP_DI".DB91_DBX063_6;
      CLR;
      =     "MAP_DI".DB91_DBX063_7;
NETWORK
TITLE = da DB91.dbx64.0 a DB91.dbx64.7
      CLR;
      =     "MAP_DI".DB91_DBX064_0;
      =     "MAP_DI".DB91_DBX064_1;
      =     "MAP_DI".DB91_DBX064_2;
      =     "MAP_DI".DB91_DBX064_3;
      =     "MAP_DI".DB91_DBX064_4;
      =     "MAP_DI".DB91_DBX064_5;
      A     "-488Y8";
      =     "MAP_DI".DB91_DBX064_6;
      A     "-465S8";
      =     "MAP_DI".DB91_DBX064_7;
NETWORK
TITLE = da DB91.dbx65.0 a DB91.dbx65.7
      A     "-466S1";
      =     "MAP_DI".DB91_DBX065_0;
      A     "-466S2";
      =     "MAP_DI".DB91_DBX065_1;
      CLR;
      =     "MAP_DI".DB91_DBX065_2;
      =     "MAP_DI".DB91_DBX065_3;
      =     "MAP_DI".DB91_DBX065_4;
      =     "MAP_DI".DB91_DBX065_5;
      =     "MAP_DI".DB91_DBX065_6;
      =     "MAP_DI".DB91_DBX065_7;
NETWORK
TITLE = da DB91.dbx66.0 a DB91.dbx66.7
      L     B#16#0;
      T     DB91.DBB 66;
NETWORK
TITLE = da DB91.dbx67.0 a DB91.dbx67.7
      A     "-468S5";
      =     "MAP_DI".DB91_DBX067_0;
      A     "-468S6";
      =     "MAP_DI".DB91_DBX067_1;
      A     "-468S7";
      =     "MAP_DI".DB91_DBX067_2;
      A     "-468S8";
      =     "MAP_DI".DB91_DBX067_3;
      CLR;
      =     "MAP_DI".DB91_DBX067_4;
      =     "MAP_DI".DB91_DBX067_5;
      =     "MAP_DI".DB91_DBX067_6;
      =     "MAP_DI".DB91_DBX067_7;
NETWORK
TITLE = da DB91.dbx68.0 a DB91.dbx68.7
      L     B#16#0;
      T     DB91.DBB 68;
NETWORK
TITLE = da DB91.dbx69.0 a DB91.dbx69.7
      L     B#16#0;
      T     DB91.DBB 69;
NETWORK
TITLE = da DB91.dbx70.0 a DB91.dbx70.7
      A     "-467B1";
      =     "MAP_DI".DB91_DBX070_0;
      A     "-467B2";
      =     "MAP_DI".DB91_DBX070_1;
      A     "-467B3";
      =     "MAP_DI".DB91_DBX070_2;
      A     "-467B4";
      =     "MAP_DI".DB91_DBX070_3;
      A     "-467B5";
      =     "MAP_DI".DB91_DBX070_4;
      A     "-467B6";
      =     "MAP_DI".DB91_DBX070_5;
      A     "-467B7";
      =     "MAP_DI".DB91_DBX070_6;
      A     "-467B8";
      =     "MAP_DI".DB91_DBX070_7;
NETWORK
TITLE = da DB91.dbx71.0 a DB91.dbx71.7
      A     "-468B1";
      =     "MAP_DI".DB91_DBX071_0;
      A     "-468B2";
      =     "MAP_DI".DB91_DBX071_1;
      A     "-468B3";
      =     "MAP_DI".DB91_DBX071_2;
      A     "-468B4";
      =     "MAP_DI".DB91_DBX071_3;
      CLR;
      =     "MAP_DI".DB91_DBX071_4;
      =     "MAP_DI".DB91_DBX071_5;
      =     "MAP_DI".DB91_DBX071_6;
      =     "MAP_DI".DB91_DBX071_7;
NETWORK
TITLE = da DB91.dbx72.0 a DB91.dbx72.7
      L     B#16#0;
      T     DB91.DBB 72;
NETWORK
TITLE = da DB91.dbx73.0 a DB91.dbx73.7
      L     B#16#0;
      T     DB91.DBB 73;
NETWORK
TITLE = da DB91.dbx74.0 a DB91.dbx74.7
      L     B#16#0;
      T     DB91.DBB 74;
NETWORK
TITLE = da DB91.dbx75.0 a DB91.dbx75.7
      L     B#16#0;
      T     DB91.DBB 75;
NETWORK
TITLE = da DB91.dbx76.0 a DB91.dbx76.7
      A     "+MCB12:7";
      =     "MAP_DI".DB91_DBX076_0;
      A     "+MCB12:8";
      =     "MAP_DI".DB91_DBX076_1;
      A     "+MCB12:9";
      =     "MAP_DI".DB91_DBX076_2;
      A     "+MCB12:10";
      =     "MAP_DI".DB91_DBX076_3;
      CLR;
      =     "MAP_DI".DB91_DBX076_4;
      =     "MAP_DI".DB91_DBX076_5;
      =     "MAP_DI".DB91_DBX076_6;
      =     "MAP_DI".DB91_DBX076_7;
NETWORK
TITLE = da DB91.dbx77.0 a DB91.dbx77.7
      A     "-475S2/S2A";
      =     "MAP_DI".DB91_DBX077_0;
      A     "-475S1/S1A";
      =     "MAP_DI".DB91_DBX077_1;
      CLR;
      =     "MAP_DI".DB91_DBX077_2;
      =     "MAP_DI".DB91_DBX077_3;
      =     "MAP_DI".DB91_DBX077_4;
      =     "MAP_DI".DB91_DBX077_5;
      =     "MAP_DI".DB91_DBX077_6;
      =     "MAP_DI".DB91_DBX077_7;
NETWORK
TITLE = da DB91.dbx78.0 a DB91.dbx78.7
      CLR;
      =     "MAP_DI".DB91_DBX078_0;
      =     "MAP_DI".DB91_DBX078_1;
      A     "-340Q1";
      =     "MAP_DI".DB91_DBX078_2;
      A     "-109Q9";
      =     "MAP_DI".DB91_DBX078_3;
      A     "-305Q2";
      =     "MAP_DI".DB91_DBX078_4;
      A     "-305Q1";
      =     "MAP_DI".DB91_DBX078_5;
      CLR;
      =     "MAP_DI".DB91_DBX078_6;
      A     "-306Q1";
      =     "MAP_DI".DB91_DBX078_7;
NETWORK
TITLE = da DB91.dbx79.0 a DB91.dbx79.7
      L     B#16#0;
      T     DB91.DBB 79;
NETWORK
TITLE = da DB91.dbx80.0 a DB91.dbx80.7
      A     "-361S1";
      =     "MAP_DI".DB91_DBX080_0;
      A     "-361S2";
      =     "MAP_DI".DB91_DBX080_1;
      A     "-361S3";
      =     "MAP_DI".DB91_DBX080_2;
      A     "-361S4";
      =     "MAP_DI".DB91_DBX080_3;
      A     "-361S5";
      =     "MAP_DI".DB91_DBX080_4;
      A     "-361B6";
      =     "MAP_DI".DB91_DBX080_5;
      A     "-361B7";
      =     "MAP_DI".DB91_DBX080_6;
      A     "-361S8";
      =     "MAP_DI".DB91_DBX080_7;
NETWORK
TITLE = da DB91.dbx81.0 a DB91.dbx81.7
      A     "-361B1";
      =     "MAP_DI".DB91_DBX081_0;
      A     "-362B2";
      =     "MAP_DI".DB91_DBX081_1;
      A     "-362S3";
      =     "MAP_DI".DB91_DBX081_2;
      A     "-386Y1";
      =     "MAP_DI".DB91_DBX081_3;
      A     "-362S5";
      =     "MAP_DI".DB91_DBX081_4;
      A     "-362S6";
      =     "MAP_DI".DB91_DBX081_5;
      A     "-362B7";
      =     "MAP_DI".DB91_DBX081_6;
      A     "-362B8";
      =     "MAP_DI".DB91_DBX081_7;
NETWORK
TITLE = da DB91.dbx82.0 a DB91.dbx82.7
      A     "-363S1";
      =     "MAP_DI".DB91_DBX082_0;
      A     "-363S2";
      =     "MAP_DI".DB91_DBX082_1;
      A     "-363S3";
      =     "MAP_DI".DB91_DBX082_2;
      A     "-363S4";
      =     "MAP_DI".DB91_DBX082_3;
      A     "-363S5:CLOSING";
      =     "MAP_DI".DB91_DBX082_4;
      A     "-363S5:OPENING";
      =     "MAP_DI".DB91_DBX082_5;
      A     "-363S7:CLOSING";
      =     "MAP_DI".DB91_DBX082_6;
      A     "-363S7:OPENING";
      =     "MAP_DI".DB91_DBX082_7;
NETWORK
TITLE = da DB91.dbx83.0 a DB91.dbx83.7
      A     "-364S1:Closing";
      =     "MAP_DI".DB91_DBX083_0;
      A     "-364S1:Opening";
      =     "MAP_DI".DB91_DBX083_1;
      CLR;
      =     "MAP_DI".DB91_DBX083_2;
      =     "MAP_DI".DB91_DBX083_3;
      =     "MAP_DI".DB91_DBX083_4;
      =     "MAP_DI".DB91_DBX083_5;
      A     "-364S7";
      =     "MAP_DI".DB91_DBX083_6;
      CLR;
      =     "MAP_DI".DB91_DBX083_7;
NETWORK
TITLE = da DB91.dbx84.0 a DB91.dbx84.7
      CLR;
      =     "MAP_DI".DB91_DBX084_0;
      =     "MAP_DI".DB91_DBX084_1;
      =     "MAP_DI".DB91_DBX084_2;
      =     "MAP_DI".DB91_DBX084_3;
      =     "MAP_DI".DB91_DBX084_4;
      =     "MAP_DI".DB91_DBX084_5;
      A     "-388Y8";
      =     "MAP_DI".DB91_DBX084_6;
      CLR;
      =     "MAP_DI".DB91_DBX084_7;
NETWORK
TITLE = da DB91.dbx85.0 a DB91.dbx85.7
      A     "-365S";
      =     "MAP_DI".DB91_DBX085_0;
      A     "-366S1";
      =     "MAP_DI".DB91_DBX085_1;
      CLR;
      =     "MAP_DI".DB91_DBX085_2;
      =     "MAP_DI".DB91_DBX085_3;
      =     "MAP_DI".DB91_DBX085_4;
      =     "MAP_DI".DB91_DBX085_5;
      =     "MAP_DI".DB91_DBX085_6;
      =     "MAP_DI".DB91_DBX085_7;
NETWORK
TITLE = da DB91.dbx86.0 a DB91.dbx86.7
      L     B#16#0;
      T     DB91.DBB 86;
NETWORK
TITLE = da DB91.dbx87.0 a DB91.dbx87.7
      A     "-367S7";
      =     "MAP_DI".DB91_DBX087_0;
      A     "-367S8";
      =     "MAP_DI".DB91_DBX087_1;
      A     "-368S1";
      =     "MAP_DI".DB91_DBX087_2;
      A     "-368S2";
      =     "MAP_DI".DB91_DBX087_3;
      CLR;
      =     "MAP_DI".DB91_DBX087_4;
      =     "MAP_DI".DB91_DBX087_5;
      =     "MAP_DI".DB91_DBX087_6;
      =     "MAP_DI".DB91_DBX087_7;
NETWORK
TITLE = DB91.dbx88.0 a DB91.dbx68.7
      L     B#16#0;
      T     DB91.DBB 88;
NETWORK
TITLE = da DB91.dbx89.0 a DB91.dbx69.7
      L     B#16#0;
      T     DB91.DBB 89;
NETWORK
TITLE = da DB91.dbx90.0 a DB91.dbx90.7
      A     "-367B1";
      =     "MAP_DI".DB91_DBX090_0;
      A     "-367B2";
      =     "MAP_DI".DB91_DBX090_1;
      A     "-367B3";
      =     "MAP_DI".DB91_DBX090_2;
      A     "-367B4";
      =     "MAP_DI".DB91_DBX090_3;
      A     "-367B5";
      =     "MAP_DI".DB91_DBX090_4;
      A     "-367B6";
      =     "MAP_DI".DB91_DBX090_5;
      CLR;
      =     "MAP_DI".DB91_DBX090_6;
      CLR;
      =     "MAP_DI".DB91_DBX090_7;
NETWORK
TITLE = da DB91.dbx91.0 a DB91.dbx91.7
      L     B#16#0;
      T     DB91.DBB 91;
NETWORK
TITLE = da DB91.dbx92.0 a DB91.dbx92.7
      L     B#16#0;
      T     DB91.DBB 92;
NETWORK
TITLE = da DB91.dbx93.0 a DB91.dbx93.7
      L     B#16#0;
      T     DB91.DBB 93;
NETWORK
TITLE = da DB91.dbx94.0 a DB91.dbx94.7
      L     B#16#0;
      T     DB91.DBB 94;
NETWORK
TITLE = da DB91.dbx95.0 a DB91.dbx95.7
      L     B#16#0;
      T     DB91.DBB 95;
NETWORK
TITLE = da DB91.dbx96.0 a DB91.dbx96.7
      A     "+MCB06:7";
      =     "MAP_DI".DB91_DBX096_0;
      A     "+MCB06:8";
      =     "MAP_DI".DB91_DBX096_1;
      A     "+MCB06:9";
      =     "MAP_DI".DB91_DBX096_2;
      A     "+MCB06:10";
      =     "MAP_DI".DB91_DBX096_3;
      CLR;
      =     "MAP_DI".DB91_DBX096_4;
      =     "MAP_DI".DB91_DBX096_5;
      =     "MAP_DI".DB91_DBX096_6;
      =     "MAP_DI".DB91_DBX096_7;
NETWORK
TITLE = da DB91.dbx97.0 a DB91.dbx97.7
      A     "-375S7/S7A";
      =     "MAP_DI".DB91_DBX097_0;
      A     "-374S7/S7A";
      =     "MAP_DI".DB91_DBX097_1;
      CLR;
      =     "MAP_DI".DB91_DBX097_2;
      =     "MAP_DI".DB91_DBX097_3;
      =     "MAP_DI".DB91_DBX097_4;
      =     "MAP_DI".DB91_DBX097_5;
      =     "MAP_DI".DB91_DBX097_6;
      =     "MAP_DI".DB91_DBX097_7;
NETWORK
TITLE = da DB91.dbx98.0 a DB91.dbx98.7
      L     B#16#0;
      T     DB91.DBB 98;
NETWORK
TITLE = da DB91.dbx99.0 a DB91.dbx99.7
      A     "-375S1";
      =     "MAP_DI".DB91_DBX099_0;
      A     "-375B1";
      =     "MAP_DI".DB91_DBX099_1;
      A     "-375S3";
      =     "MAP_DI".DB91_DBX099_2;
      A     "-375S4";
      =     "MAP_DI".DB91_DBX099_3;
      A     "-375S5";
      =     "MAP_DI".DB91_DBX099_4;
      CLR;
      =     "MAP_DI".DB91_DBX099_5;
      =     "MAP_DI".DB91_DBX099_6;
      =     "MAP_DI".DB91_DBX099_7;
END_FUNCTION

FUNCTION "Map Output Function" : VOID	// FC 93
TITLE = MAP OUTPUT FUNCTION
VERSION : 0.1
VAR_TEMP
  Temp1 : BOOL ;
END_VAR
BEGIN
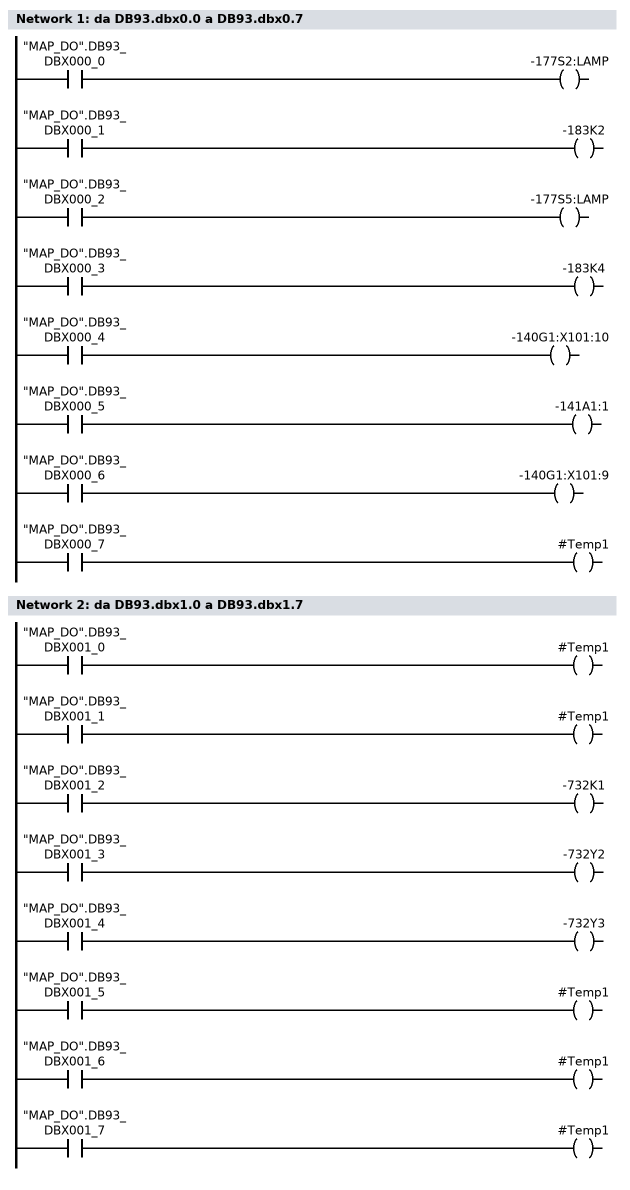
NETWORK
TITLE = da DB93.dbx0.0 a DB93.dbx0.7
      A     "MAP_DO".DB93_DBX000_0;
      =     "-177S2:LAMP";
      A     "MAP_DO".DB93_DBX000_1;
      =     "-183K2";
      A     "MAP_DO".DB93_DBX000_2;
      =     "-177S5:LAMP";
      A     "MAP_DO".DB93_DBX000_3;
      =     "-183K4";
      A     "MAP_DO".DB93_DBX000_4;
      =     "-140G1:X101:10";
      A     "MAP_DO".DB93_DBX000_5;
      =     "-141A1:1";
      A     "MAP_DO".DB93_DBX000_6;
      =     "-140G1:X101:9";
      A     "MAP_DO".DB93_DBX000_7;
      =     #Temp1;
NETWORK
TITLE = da DB93.dbx1.0 a DB93.dbx1.7
      A     "MAP_DO".DB93_DBX001_0;
      =     #Temp1;
      A     "MAP_DO".DB93_DBX001_1;
      =     #Temp1;
      A     "MAP_DO".DB93_DBX001_2;
      =     "-732K1";
      A     "MAP_DO".DB93_DBX001_3;
      =     "-732Y2";
      A     "MAP_DO".DB93_DBX001_4;
      =     "-732Y3";
      A     "MAP_DO".DB93_DBX001_5;
      =     #Temp1;
      A     "MAP_DO".DB93_DBX001_6;
      =     #Temp1;
      A     "MAP_DO".DB93_DBX001_7;
      =     #Temp1;
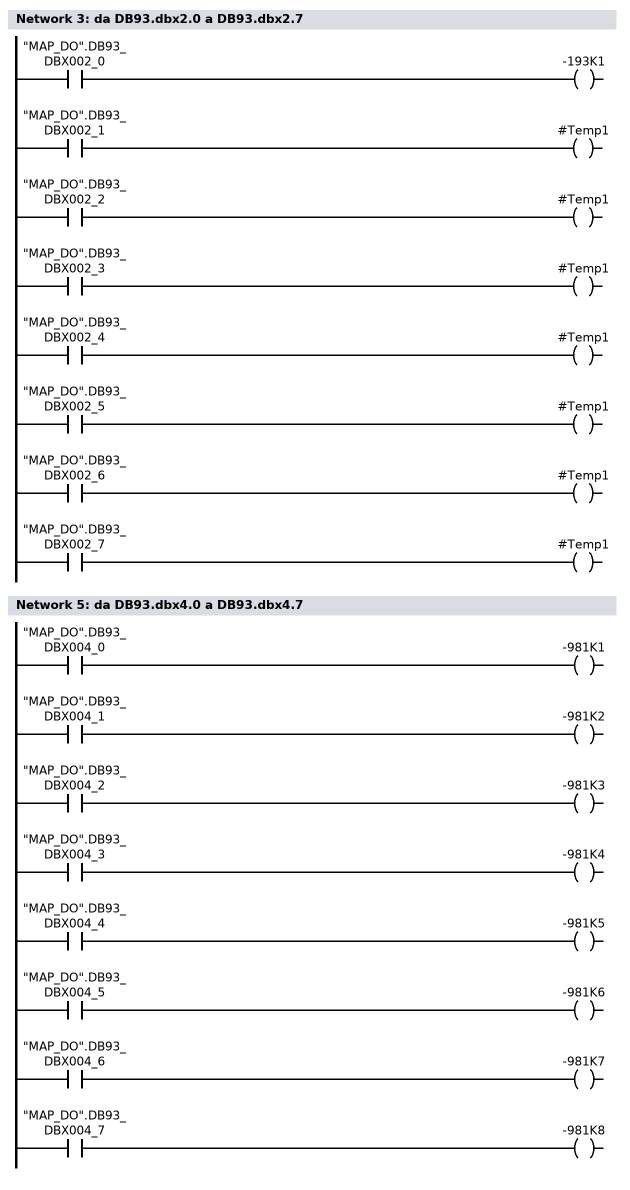
NETWORK
TITLE = da DB93.dbx2.0 a DB93.dbx2.7
      A     "MAP_DO".DB93_DBX002_0;
      =     "-193K1";
      A     "MAP_DO".DB93_DBX002_1;
      =     #Temp1;
      A     "MAP_DO".DB93_DBX002_2;
      =     #Temp1;
      A     "MAP_DO".DB93_DBX002_3;
      =     #Temp1;
      A     "MAP_DO".DB93_DBX002_4;
      =     #Temp1;
      A     "MAP_DO".DB93_DBX002_5;
      =     #Temp1;
      A     "MAP_DO".DB93_DBX002_6;
      =     #Temp1;
      A     "MAP_DO".DB93_DBX002_7;
      =     #Temp1;
NETWORK
TITLE = da DB93.dbx3.0 a DB93.dbx3.7
NETWORK
TITLE = da DB93.dbx4.0 a DB93.dbx4.7
      A     "MAP_DO".DB93_DBX004_0;
      =     "-981K1";
      A     "MAP_DO".DB93_DBX004_1;
      =     "-981K2";
      A     "MAP_DO".DB93_DBX004_2;
      =     "-981K3";
      A     "MAP_DO".DB93_DBX004_3;
      =     "-981K4";
      A     "MAP_DO".DB93_DBX004_4;
      =     "-981K5";
      A     "MAP_DO".DB93_DBX004_5;
      =     "-981K6";
      A     "MAP_DO".DB93_DBX004_6;
      =     "-981K7";
      A     "MAP_DO".DB93_DBX004_7;
      =     "-981K8";
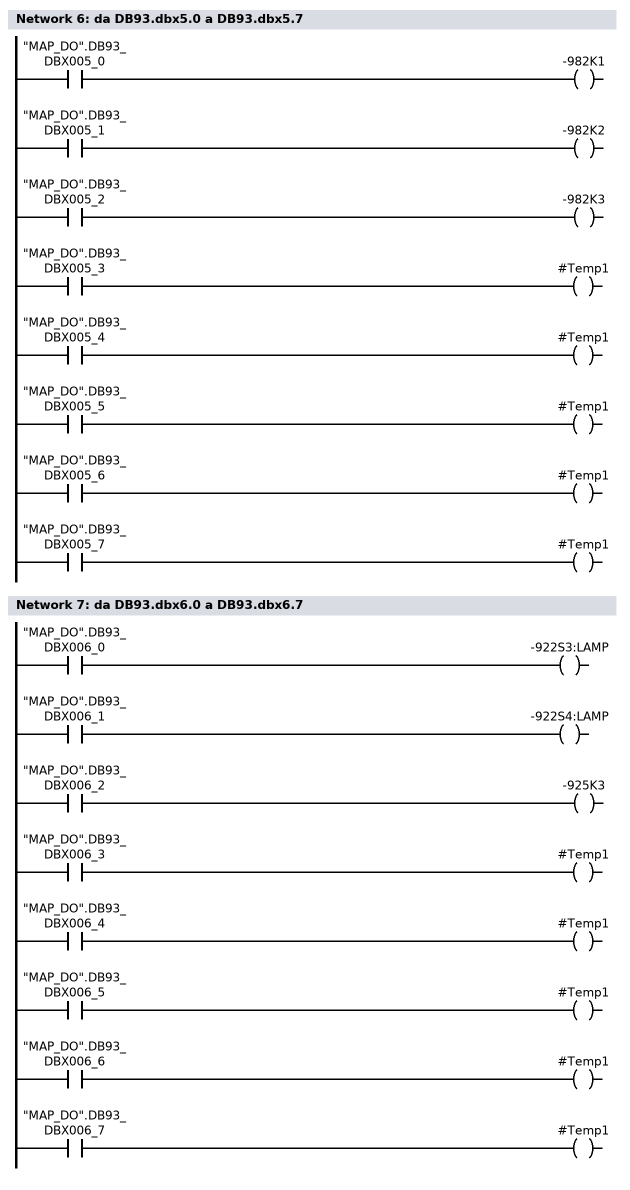
NETWORK
TITLE = da DB93.dbx5.0 a DB93.dbx5.7
      A     "MAP_DO".DB93_DBX005_0;
      =     "-982K1";
      A     "MAP_DO".DB93_DBX005_1;
      =     "-982K2";
      A     "MAP_DO".DB93_DBX005_2;
      =     "-982K3";
      A     "MAP_DO".DB93_DBX005_3;
      =     #Temp1;
      A     "MAP_DO".DB93_DBX005_4;
      =     #Temp1;
      A     "MAP_DO".DB93_DBX005_5;
      =     #Temp1;
      A     "MAP_DO".DB93_DBX005_6;
      =     #Temp1;
      A     "MAP_DO".DB93_DBX005_7;
      =     #Temp1;
NETWORK
TITLE = da DB93.dbx6.0 a DB93.dbx6.7
      A     "MAP_DO".DB93_DBX006_0;
      =     "-922S3:LAMP";
      A     "MAP_DO".DB93_DBX006_1;
      =     "-922S4:LAMP";
      A     "MAP_DO".DB93_DBX006_2;
      =     "-925K3";
      A     "MAP_DO".DB93_DBX006_3;
      =     #Temp1;
      A     "MAP_DO".DB93_DBX006_4;
      =     #Temp1;
      A     "MAP_DO".DB93_DBX006_5;
      =     #Temp1;
      A     "MAP_DO".DB93_DBX006_6;
      =     #Temp1;
      A     "MAP_DO".DB93_DBX006_7;
      =     #Temp1;
NETWORK
TITLE = da DB93.dbx7.0 a DB93.dbx7.7
NETWORK
TITLE = da DB93.dbx8.0 a DB93.dbx8.7
NETWORK
TITLE = da DB93.dbx9.0 a DB93.dbx9.7
NETWORK
TITLE = da DB93.dbx10.0 a DB93.dbx10.7
NETWORK
TITLE = da DB93.dbx11.0 a DB93.dbx11.7
NETWORK
TITLE = da DB93.dbx12.0 a DB93.dbx12.7
NETWORK
TITLE = da DB93.dbx13.0 a DB93.dbx13.7
NETWORK
TITLE = da DB93.dbx14.0 a DB93.dbx14.7
NETWORK
TITLE = da DB93.dbx15.0 a DB93.dbx15.7
NETWORK
TITLE = da DB93.dbx16.0 a DB93.dbx16.7
NETWORK
TITLE = da DB93.dbx17.0 a DB93.dbx17.7
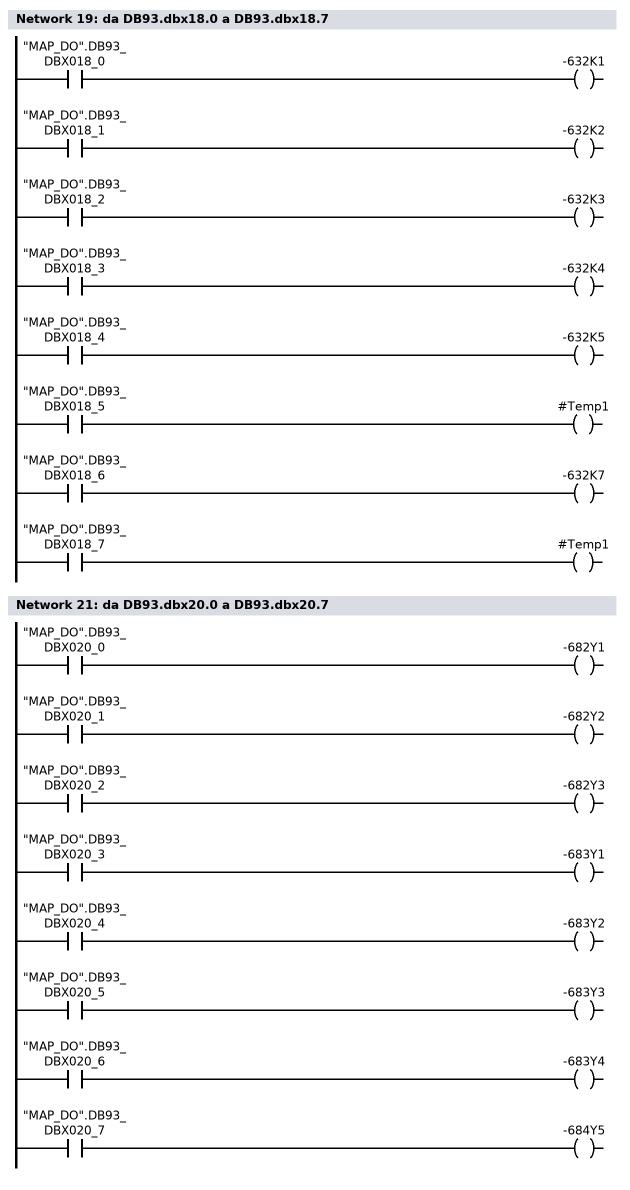
NETWORK
TITLE = da DB93.dbx18.0 a DB93.dbx18.7
      A     "MAP_DO".DB93_DBX018_0;
      =     "-632K1";
      A     "MAP_DO".DB93_DBX018_1;
      =     "-632K2";
      A     "MAP_DO".DB93_DBX018_2;
      =     "-632K3";
      A     "MAP_DO".DB93_DBX018_3;
      =     "-632K4";
      A     "MAP_DO".DB93_DBX018_4;
      =     "-632K5";
      A     "MAP_DO".DB93_DBX018_5;
      =     #Temp1;
      A     "MAP_DO".DB93_DBX018_6;
      =     "-632K7";
      A     "MAP_DO".DB93_DBX018_7;
      =     #Temp1;
NETWORK
TITLE = da DB93.dbx19.0 a DB93.dbx19.7
NETWORK
TITLE = da DB93.dbx20.0 a DB93.dbx20.7
      A     "MAP_DO".DB93_DBX020_0;
      =     "-682Y1";
      A     "MAP_DO".DB93_DBX020_1;
      =     "-682Y2";
      A     "MAP_DO".DB93_DBX020_2;
      =     "-682Y3";
      A     "MAP_DO".DB93_DBX020_3;
      =     "-683Y1";
      A     "MAP_DO".DB93_DBX020_4;
      =     "-683Y2";
      A     "MAP_DO".DB93_DBX020_5;
      =     "-683Y3";
      A     "MAP_DO".DB93_DBX020_6;
      =     "-683Y4";
      A     "MAP_DO".DB93_DBX020_7;
      =     "-684Y5";
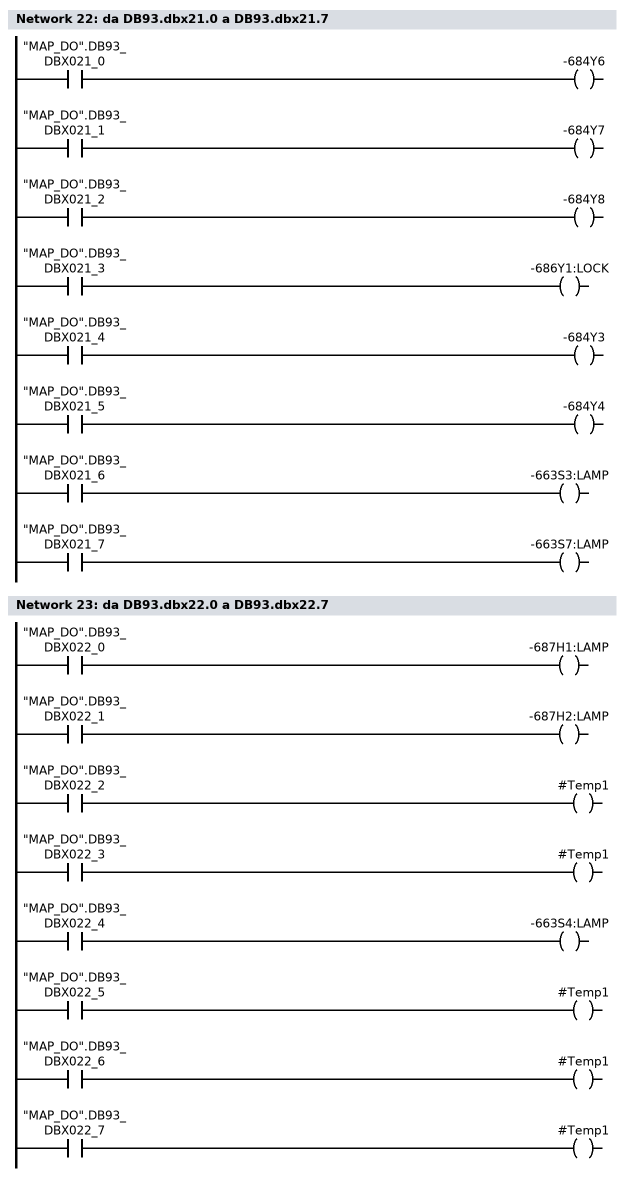
NETWORK
TITLE = da DB93.dbx21.0 a DB93.dbx21.7
      A     "MAP_DO".DB93_DBX021_0;
      =     "-684Y6";
      A     "MAP_DO".DB93_DBX021_1;
      =     "-684Y7";
      A     "MAP_DO".DB93_DBX021_2;
      =     "-684Y8";
      A     "MAP_DO".DB93_DBX021_3;
      =     "-686Y1:LOCK";
      A     "MAP_DO".DB93_DBX021_4;
      =     "-684Y3";
      A     "MAP_DO".DB93_DBX021_5;
      =     "-684Y4";
      A     "MAP_DO".DB93_DBX021_6;
      =     "-663S3:LAMP";
      A     "MAP_DO".DB93_DBX021_7;
      =     "-663S7:LAMP";
NETWORK
TITLE = da DB93.dbx22.0 a DB93.dbx22.7
      A     "MAP_DO".DB93_DBX022_0;
      =     "-687H1:LAMP";
      A     "MAP_DO".DB93_DBX022_1;
      =     "-687H2:LAMP";
      A     "MAP_DO".DB93_DBX022_2;
      =     #Temp1;
      A     "MAP_DO".DB93_DBX022_3;
      =     #Temp1;
      A     "MAP_DO".DB93_DBX022_4;
      =     "-663S4:LAMP";
      A     "MAP_DO".DB93_DBX022_5;
      =     #Temp1;
      A     "MAP_DO".DB93_DBX022_6;
      =     #Temp1;
      A     "MAP_DO".DB93_DBX022_7;
      =     #Temp1;
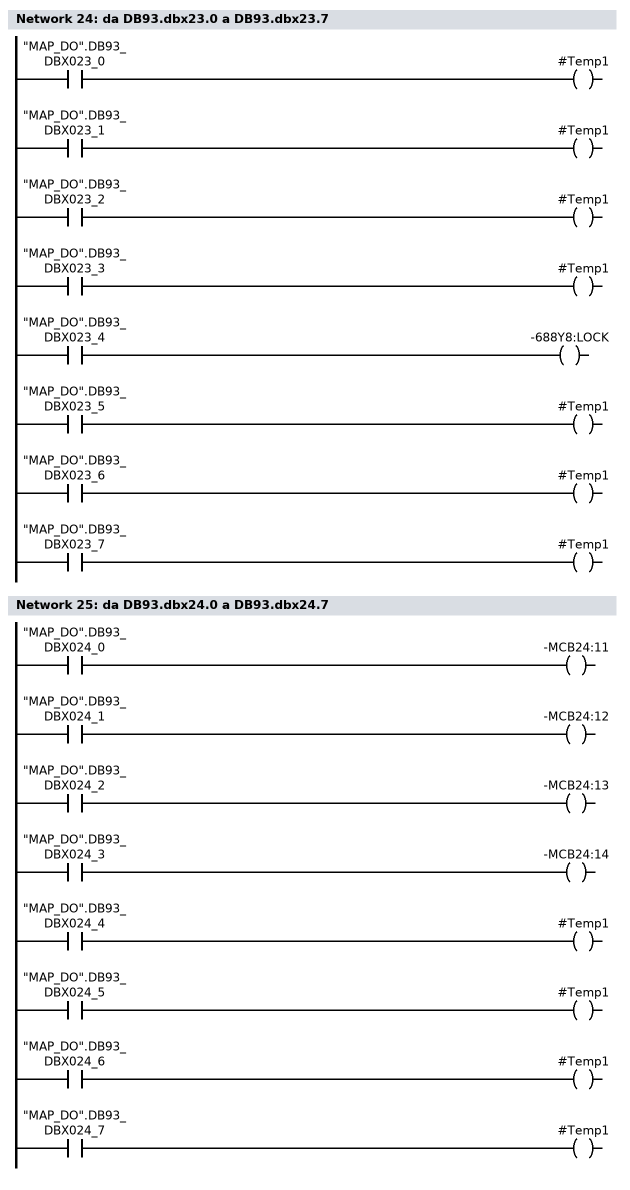
NETWORK
TITLE = da DB93.dbx23.0 a DB93.dbx23.7
      A     "MAP_DO".DB93_DBX023_0;
      =     #Temp1;
      A     "MAP_DO".DB93_DBX023_1;
      =     #Temp1;
      A     "MAP_DO".DB93_DBX023_2;
      =     #Temp1;
      A     "MAP_DO".DB93_DBX023_3;
      =     #Temp1;
      A     "MAP_DO".DB93_DBX023_4;
      =     "-688Y8:LOCK";
      A     "MAP_DO".DB93_DBX023_5;
      =     #Temp1;
      A     "MAP_DO".DB93_DBX023_6;
      =     #Temp1;
      A     "MAP_DO".DB93_DBX023_7;
      =     #Temp1;
NETWORK
TITLE = da DB93.dbx24.0 a DB93.dbx24.7
      A     "MAP_DO".DB93_DBX024_0;
      =     "-MCB24:11";
      A     "MAP_DO".DB93_DBX024_1;
      =     "-MCB24:12";
      A     "MAP_DO".DB93_DBX024_2;
      =     "-MCB24:13";
      A     "MAP_DO".DB93_DBX024_3;
      =     "-MCB24:14";
      A     "MAP_DO".DB93_DBX024_4;
      =     #Temp1;
      A     "MAP_DO".DB93_DBX024_5;
      =     #Temp1;
      A     "MAP_DO".DB93_DBX024_6;
      =     #Temp1;
      A     "MAP_DO".DB93_DBX024_7;
      =     #Temp1;
NETWORK
TITLE = da DB93.dbx25.0 a DB93.dbx25.7
      A     "MAP_DO".DB93_DBX025_0;
      CLR;
      =     "-688Y1";
      A     "MAP_DO".DB93_DBX025_1;
      CLR;
      =     "-688Y2";
      A     "MAP_DO".DB93_DBX025_2;
      =     #Temp1;
      A     "MAP_DO".DB93_DBX025_3;
      =     #Temp1;
      A     "MAP_DO".DB93_DBX025_4;
      =     #Temp1;
      A     "MAP_DO".DB93_DBX025_5;
      =     #Temp1;
      A     "MAP_DO".DB93_DBX025_6;
      =     #Temp1;
      A     "MAP_DO".DB93_DBX025_7;
      =     #Temp1;
NETWORK
TITLE = da DB93.dbx26.0 a DB93.dbx26.7
NETWORK
TITLE = da DB93.dbx27.0 a DB93.dbx27.7
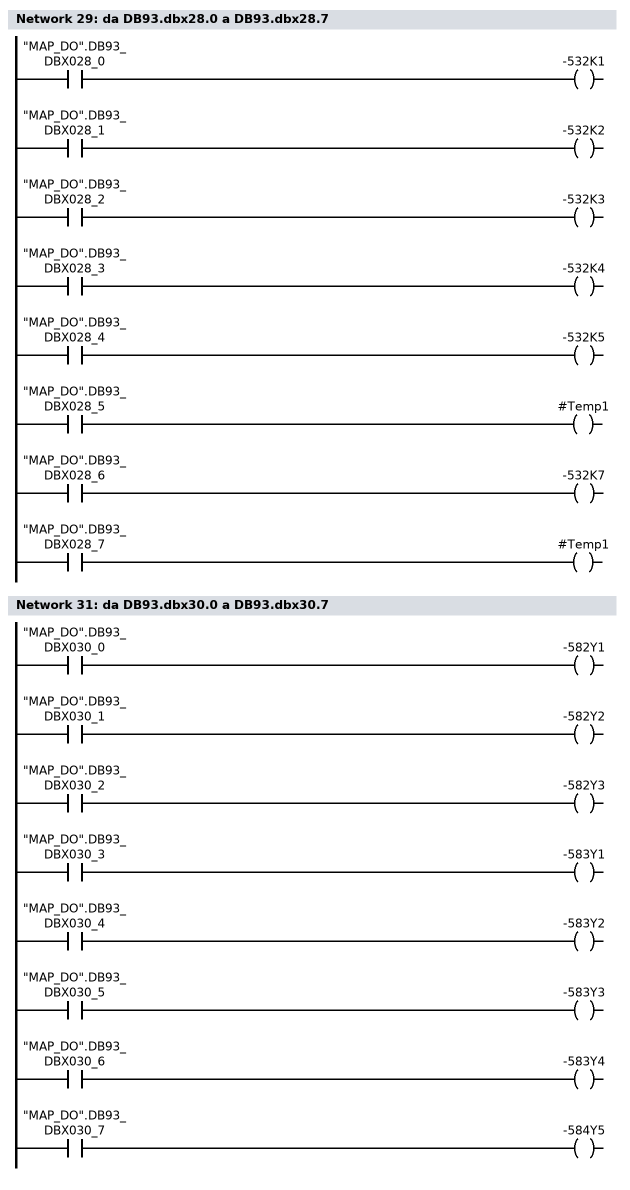
NETWORK
TITLE = da DB93.dbx28.0 a DB93.dbx28.7
      A     "MAP_DO".DB93_DBX028_0;
      =     "-532K1";
      A     "MAP_DO".DB93_DBX028_1;
      =     "-532K2";
      A     "MAP_DO".DB93_DBX028_2;
      =     "-532K3";
      A     "MAP_DO".DB93_DBX028_3;
      =     "-532K4";
      A     "MAP_DO".DB93_DBX028_4;
      =     "-532K5";
      A     "MAP_DO".DB93_DBX028_5;
      =     #Temp1;
      A     "MAP_DO".DB93_DBX028_6;
      =     "-532K7";
      A     "MAP_DO".DB93_DBX028_7;
      =     #Temp1;
NETWORK
TITLE = da DB93.dbx29.0 a DB93.dbx29.7
NETWORK
TITLE = da DB93.dbx30.0 a DB93.dbx30.7
      A     "MAP_DO".DB93_DBX030_0;
      =     "-582Y1";
      A     "MAP_DO".DB93_DBX030_1;
      =     "-582Y2";
      A     "MAP_DO".DB93_DBX030_2;
      =     "-582Y3";
      A     "MAP_DO".DB93_DBX030_3;
      =     "-583Y1";
      A     "MAP_DO".DB93_DBX030_4;
      =     "-583Y2";
      A     "MAP_DO".DB93_DBX030_5;
      =     "-583Y3";
      A     "MAP_DO".DB93_DBX030_6;
      =     "-583Y4";
      A     "MAP_DO".DB93_DBX030_7;
      =     "-584Y5";
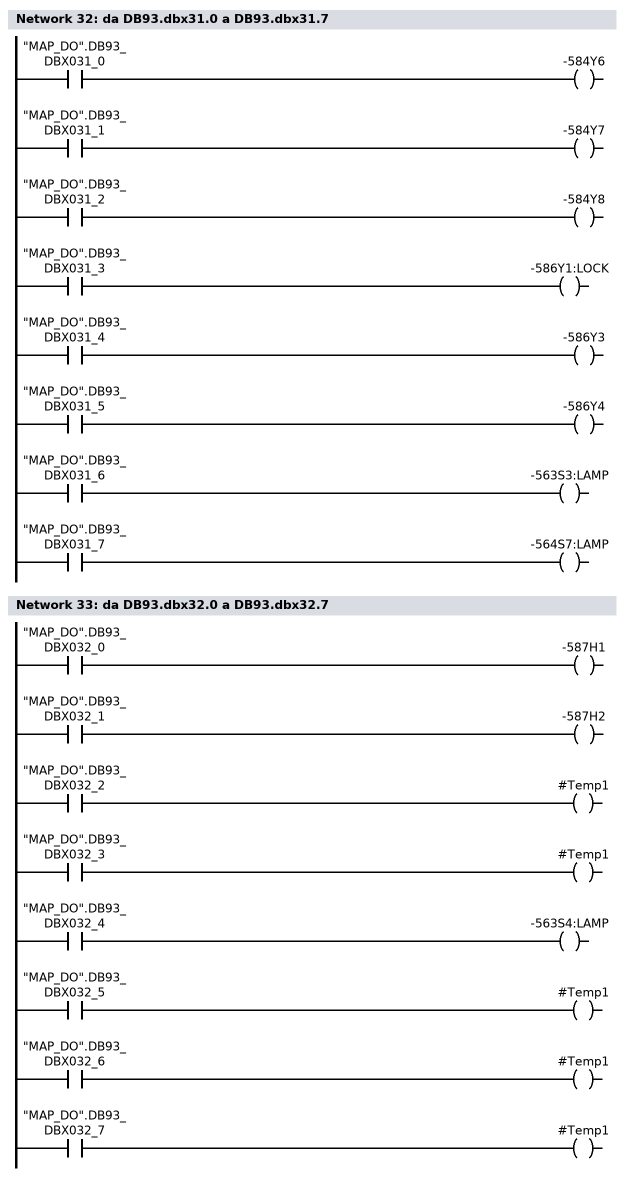
NETWORK
TITLE = da DB93.dbx31.0 a DB93.dbx31.7
      A     "MAP_DO".DB93_DBX031_0;
      =     "-584Y6";
      A     "MAP_DO".DB93_DBX031_1;
      =     "-584Y7";
      A     "MAP_DO".DB93_DBX031_2;
      =     "-584Y8";
      A     "MAP_DO".DB93_DBX031_3;
      =     "-586Y1:LOCK";
      A     "MAP_DO".DB93_DBX031_4;
      =     "-586Y3";
      A     "MAP_DO".DB93_DBX031_5;
      =     "-586Y4";
      A     "MAP_DO".DB93_DBX031_6;
      =     "-563S3:LAMP";
      A     "MAP_DO".DB93_DBX031_7;
      =     "-564S7:LAMP";
NETWORK
TITLE = da DB93.dbx32.0 a DB93.dbx32.7
      A     "MAP_DO".DB93_DBX032_0;
      =     "-587H1";
      A     "MAP_DO".DB93_DBX032_1;
      =     "-587H2";
      A     "MAP_DO".DB93_DBX032_2;
      =     #Temp1;
      A     "MAP_DO".DB93_DBX032_3;
      =     #Temp1;
      A     "MAP_DO".DB93_DBX032_4;
      =     "-563S4:LAMP";
      A     "MAP_DO".DB93_DBX032_5;
      =     #Temp1;
      A     "MAP_DO".DB93_DBX032_6;
      =     #Temp1;
      A     "MAP_DO".DB93_DBX032_7;
      =     #Temp1;
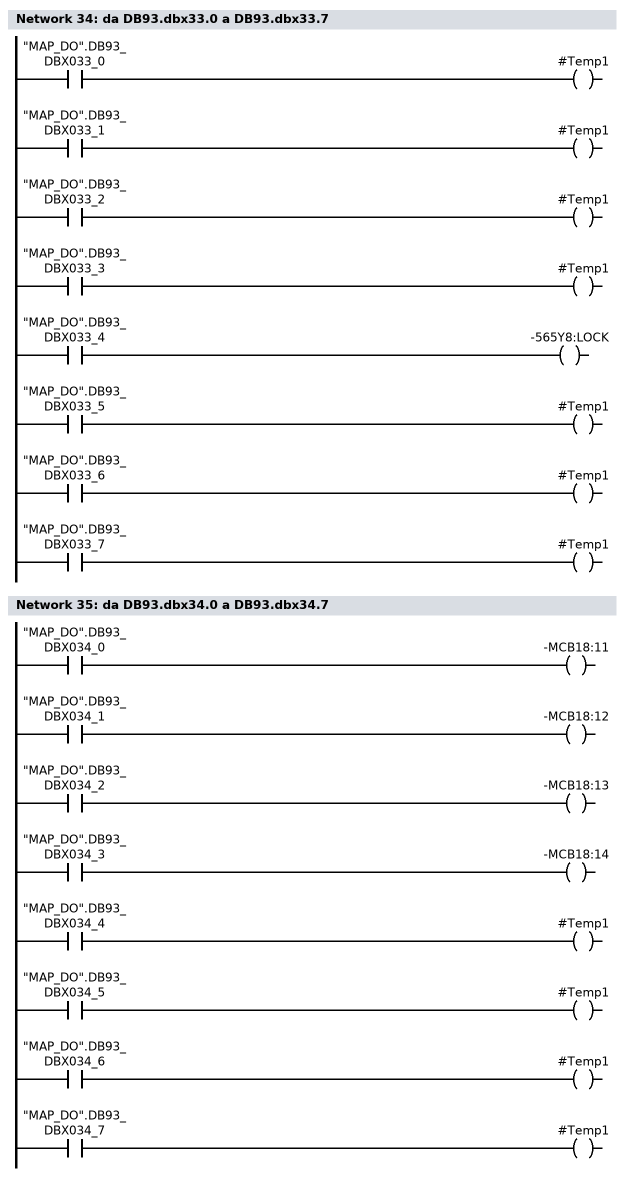
NETWORK
TITLE = da DB93.dbx33.0 a DB93.dbx33.7
      A     "MAP_DO".DB93_DBX033_0;
      =     #Temp1;
      A     "MAP_DO".DB93_DBX033_1;
      =     #Temp1;
      A     "MAP_DO".DB93_DBX033_2;
      =     #Temp1;
      A     "MAP_DO".DB93_DBX033_3;
      =     #Temp1;
      A     "MAP_DO".DB93_DBX033_4;
      =     "-565Y8:LOCK";
      A     "MAP_DO".DB93_DBX033_5;
      =     #Temp1;
      A     "MAP_DO".DB93_DBX033_6;
      =     #Temp1;
      A     "MAP_DO".DB93_DBX033_7;
      =     #Temp1;
NETWORK
TITLE = da DB93.dbx34.0 a DB93.dbx34.7
      A     "MAP_DO".DB93_DBX034_0;
      =     "-MCB18:11";
      A     "MAP_DO".DB93_DBX034_1;
      =     "-MCB18:12";
      A     "MAP_DO".DB93_DBX034_2;
      =     "-MCB18:13";
      A     "MAP_DO".DB93_DBX034_3;
      =     "-MCB18:14";
      A     "MAP_DO".DB93_DBX034_4;
      =     #Temp1;
      A     "MAP_DO".DB93_DBX034_5;
      =     #Temp1;
      A     "MAP_DO".DB93_DBX034_6;
      =     #Temp1;
      A     "MAP_DO".DB93_DBX034_7;
      =     #Temp1;
NETWORK
TITLE = da DB93.dbx35.0 a DB93.dbx35.7
      A     "MAP_DO".DB93_DBX035_0;
      CLR;
      =     "-588Y2";
      A     "MAP_DO".DB93_DBX035_1;
      CLR;
      =     "-588Y1";
      A     "MAP_DO".DB93_DBX035_2;
      =     #Temp1;
      A     "MAP_DO".DB93_DBX035_3;
      =     #Temp1;
      A     "MAP_DO".DB93_DBX035_4;
      =     #Temp1;
      A     "MAP_DO".DB93_DBX035_5;
      =     #Temp1;
      A     "MAP_DO".DB93_DBX035_6;
      =     #Temp1;
      A     "MAP_DO".DB93_DBX035_7;
      =     #Temp1;
NETWORK
TITLE = da DB93.dbx36.0 a DB93.dbx36.7
NETWORK
TITLE = da DB93.dbx37.0 a DB93.dbx37.7
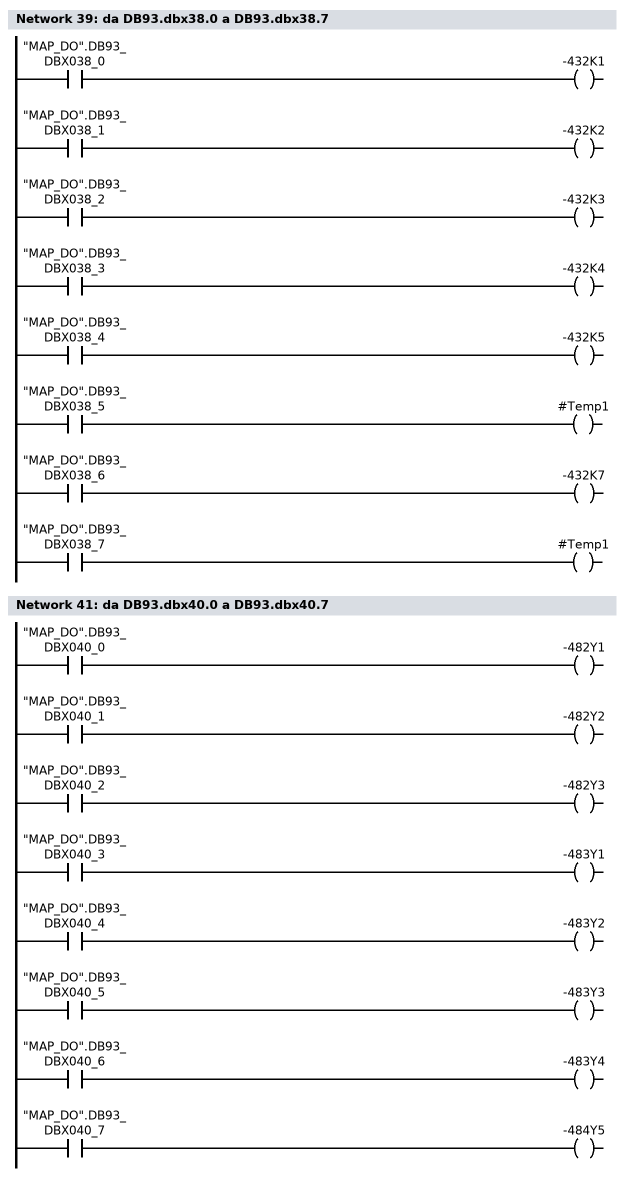
NETWORK
TITLE = da DB93.dbx38.0 a DB93.dbx38.7
      A     "MAP_DO".DB93_DBX038_0;
      =     "-432K1";
      A     "MAP_DO".DB93_DBX038_1;
      =     "-432K2";
      A     "MAP_DO".DB93_DBX038_2;
      =     "-432K3";
      A     "MAP_DO".DB93_DBX038_3;
      =     "-432K4";
      A     "MAP_DO".DB93_DBX038_4;
      =     "-432K5";
      A     "MAP_DO".DB93_DBX038_5;
      =     #Temp1;
      A     "MAP_DO".DB93_DBX038_6;
      =     "-432K7";
      A     "MAP_DO".DB93_DBX038_7;
      =     #Temp1;
NETWORK
TITLE = da DB93.dbx39.0 a DB93.dbx39.7
NETWORK
TITLE = da DB93.dbx40.0 a DB93.dbx40.7
      A     "MAP_DO".DB93_DBX040_0;
      =     "-482Y1";
      A     "MAP_DO".DB93_DBX040_1;
      =     "-482Y2";
      A     "MAP_DO".DB93_DBX040_2;
      =     "-482Y3";
      A     "MAP_DO".DB93_DBX040_3;
      =     "-483Y1";
      A     "MAP_DO".DB93_DBX040_4;
      =     "-483Y2";
      A     "MAP_DO".DB93_DBX040_5;
      =     "-483Y3";
      A     "MAP_DO".DB93_DBX040_6;
      =     "-483Y4";
      A     "MAP_DO".DB93_DBX040_7;
      =     "-484Y5";
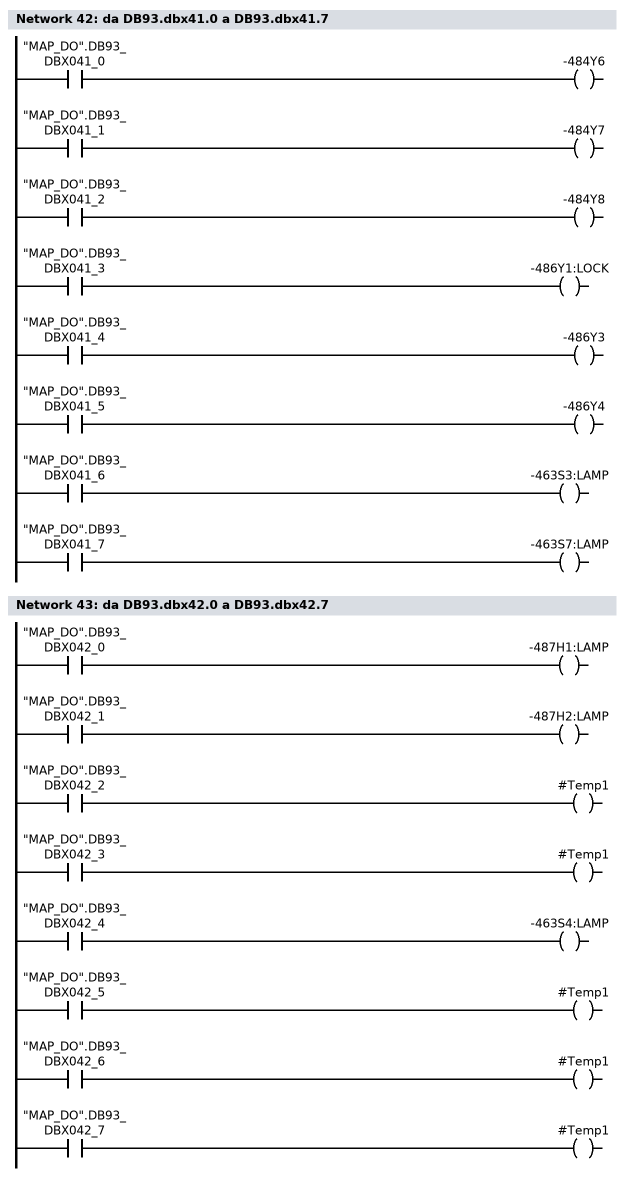
NETWORK
TITLE = da DB93.dbx41.0 a DB93.dbx41.7
      A     "MAP_DO".DB93_DBX041_0;
      =     "-484Y6";
      A     "MAP_DO".DB93_DBX041_1;
      =     "-484Y7";
      A     "MAP_DO".DB93_DBX041_2;
      =     "-484Y8";
      A     "MAP_DO".DB93_DBX041_3;
      =     "-486Y1:LOCK";
      A     "MAP_DO".DB93_DBX041_4;
      =     "-486Y3";
      A     "MAP_DO".DB93_DBX041_5;
      =     "-486Y4";
      A     "MAP_DO".DB93_DBX041_6;
      =     "-463S3:LAMP";
      A     "MAP_DO".DB93_DBX041_7;
      =     "-463S7:LAMP";
NETWORK
TITLE = da DB93.dbx42.0 a DB93.dbx42.7
      A     "MAP_DO".DB93_DBX042_0;
      =     "-487H1:LAMP";
      A     "MAP_DO".DB93_DBX042_1;
      =     "-487H2:LAMP";
      A     "MAP_DO".DB93_DBX042_2;
      =     #Temp1;
      A     "MAP_DO".DB93_DBX042_3;
      =     #Temp1;
      A     "MAP_DO".DB93_DBX042_4;
      =     "-463S4:LAMP";
      A     "MAP_DO".DB93_DBX042_5;
      =     #Temp1;
      A     "MAP_DO".DB93_DBX042_6;
      =     #Temp1;
      A     "MAP_DO".DB93_DBX042_7;
      =     #Temp1;
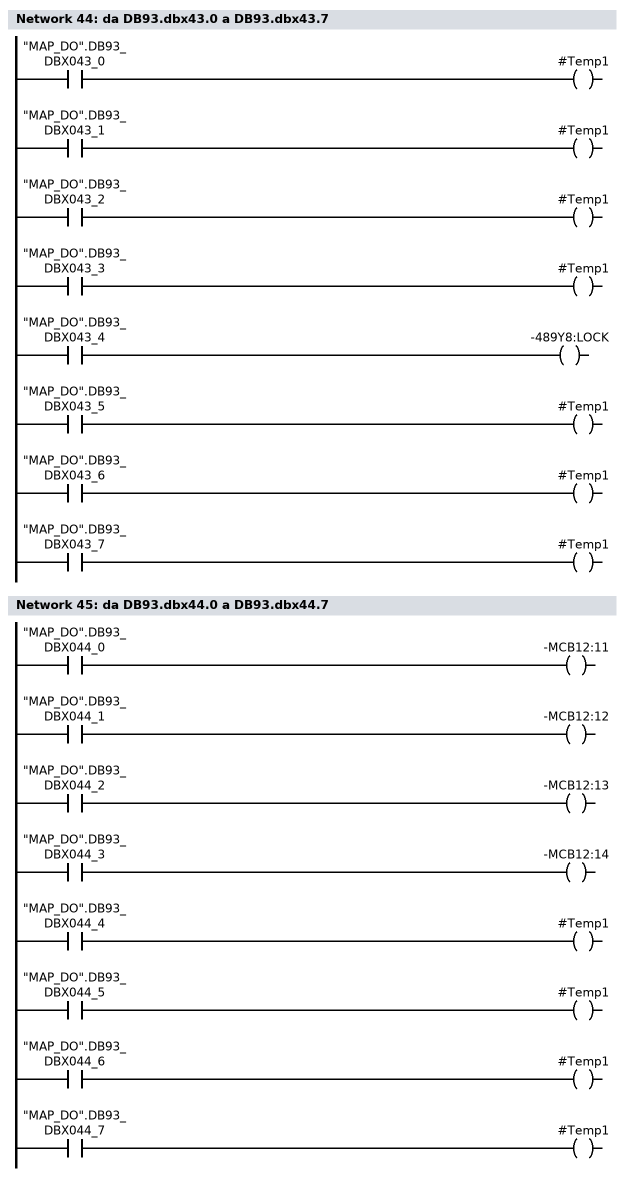
NETWORK
TITLE = da DB93.dbx43.0 a DB93.dbx43.7
      A     "MAP_DO".DB93_DBX043_0;
      =     #Temp1;
      A     "MAP_DO".DB93_DBX043_1;
      =     #Temp1;
      A     "MAP_DO".DB93_DBX043_2;
      =     #Temp1;
      A     "MAP_DO".DB93_DBX043_3;
      =     #Temp1;
      A     "MAP_DO".DB93_DBX043_4;
      =     "-489Y8:LOCK";
      A     "MAP_DO".DB93_DBX043_5;
      =     #Temp1;
      A     "MAP_DO".DB93_DBX043_6;
      =     #Temp1;
      A     "MAP_DO".DB93_DBX043_7;
      =     #Temp1;
NETWORK
TITLE = da DB93.dbx44.0 a DB93.dbx44.7
      A     "MAP_DO".DB93_DBX044_0;
      =     "-MCB12:11";
      A     "MAP_DO".DB93_DBX044_1;
      =     "-MCB12:12";
      A     "MAP_DO".DB93_DBX044_2;
      =     "-MCB12:13";
      A     "MAP_DO".DB93_DBX044_3;
      =     "-MCB12:14";
      A     "MAP_DO".DB93_DBX044_4;
      =     #Temp1;
      A     "MAP_DO".DB93_DBX044_5;
      =     #Temp1;
      A     "MAP_DO".DB93_DBX044_6;
      =     #Temp1;
      A     "MAP_DO".DB93_DBX044_7;
      =     #Temp1;
NETWORK
TITLE = da DB93.dbx45.0 a DB93.dbx45.7
      A     "MAP_DO".DB93_DBX045_0;
      CLR;
      =     "-488Y2";
      A     "MAP_DO".DB93_DBX045_1;
      CLR;
      =     "-488Y1";
      A     "MAP_DO".DB93_DBX045_2;
      =     #Temp1;
      A     "MAP_DO".DB93_DBX045_3;
      =     #Temp1;
      A     "MAP_DO".DB93_DBX045_4;
      =     #Temp1;
      A     "MAP_DO".DB93_DBX045_5;
      =     #Temp1;
      A     "MAP_DO".DB93_DBX045_6;
      =     #Temp1;
      A     "MAP_DO".DB93_DBX045_7;
      =     #Temp1;
NETWORK
TITLE = da DB93.dbx46.0 a DB93.dbx46.7
NETWORK
TITLE = da DB93.dbx47.0 a DB93.dbx47.7
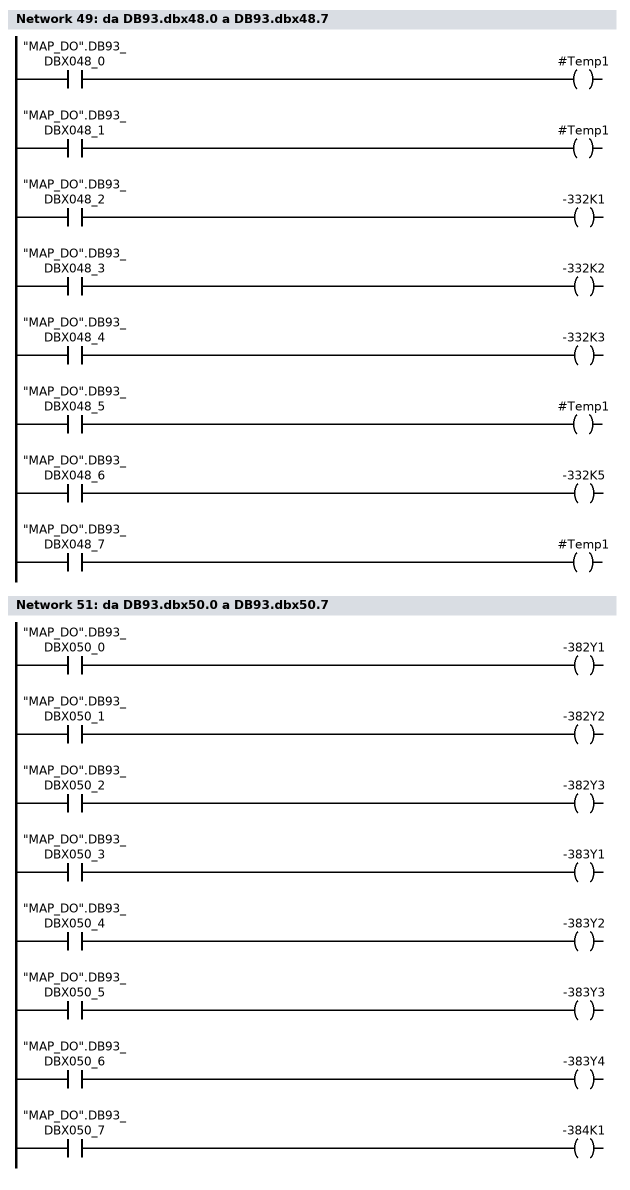
NETWORK
TITLE = da DB93.dbx48.0 a DB93.dbx48.7
      A     "MAP_DO".DB93_DBX048_0;
      =     #Temp1;
      A     "MAP_DO".DB93_DBX048_1;
      =     #Temp1;
      A     "MAP_DO".DB93_DBX048_2;
      =     "-332K1";
      A     "MAP_DO".DB93_DBX048_3;
      =     "-332K2";
      A     "MAP_DO".DB93_DBX048_4;
      =     "-332K3";
      A     "MAP_DO".DB93_DBX048_5;
      =     #Temp1;
      A     "MAP_DO".DB93_DBX048_6;
      =     "-332K5";
      A     "MAP_DO".DB93_DBX048_7;
      =     #Temp1;
NETWORK
TITLE = da DB93.dbx49.0 a DB93.dbx49.7
NETWORK
TITLE = da DB93.dbx50.0 a DB93.dbx50.7
      A     "MAP_DO".DB93_DBX050_0;
      =     "-382Y1";
      A     "MAP_DO".DB93_DBX050_1;
      =     "-382Y2";
      A     "MAP_DO".DB93_DBX050_2;
      =     "-382Y3";
      A     "MAP_DO".DB93_DBX050_3;
      =     "-383Y1";
      A     "MAP_DO".DB93_DBX050_4;
      =     "-383Y2";
      A     "MAP_DO".DB93_DBX050_5;
      =     "-383Y3";
      A     "MAP_DO".DB93_DBX050_6;
      =     "-383Y4";
      A     "MAP_DO".DB93_DBX050_7;
      =     "-384K1";
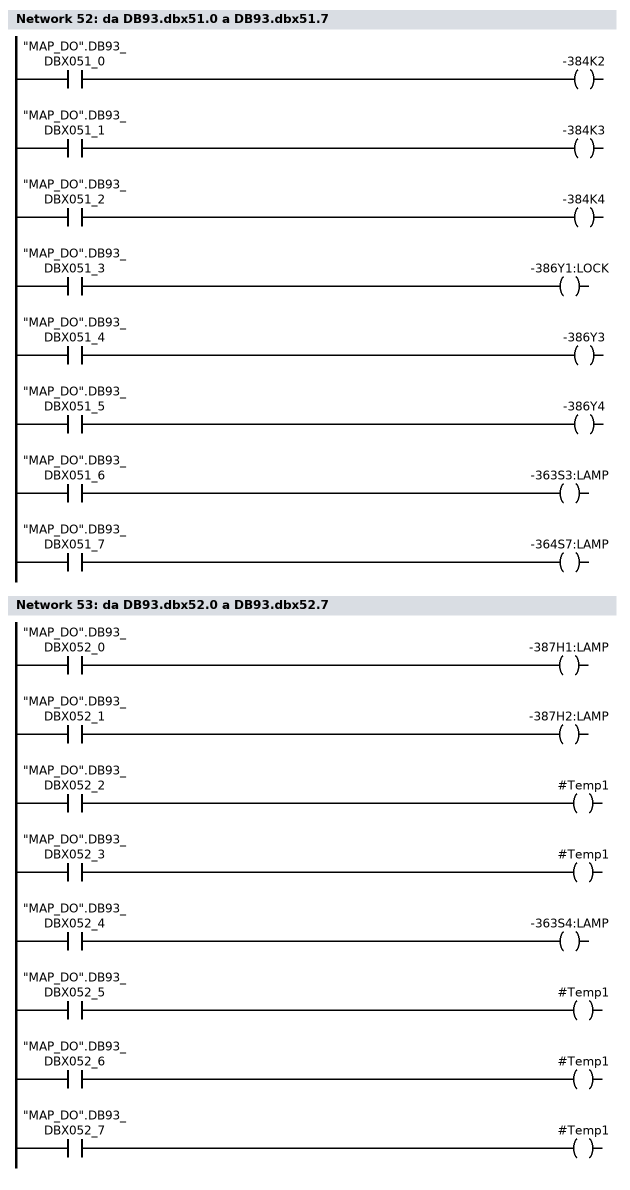
NETWORK
TITLE = da DB93.dbx51.0 a DB93.dbx51.7
      A     "MAP_DO".DB93_DBX051_0;
      =     "-384K2";
      A     "MAP_DO".DB93_DBX051_1;
      =     "-384K3";
      A     "MAP_DO".DB93_DBX051_2;
      =     "-384K4";
      A     "MAP_DO".DB93_DBX051_3;
      =     "-386Y1:LOCK";
      A     "MAP_DO".DB93_DBX051_4;
      =     "-386Y3";
      A     "MAP_DO".DB93_DBX051_5;
      =     "-386Y4";
      A     "MAP_DO".DB93_DBX051_6;
      =     "-363S3:LAMP";
      A     "MAP_DO".DB93_DBX051_7;
      =     "-364S7:LAMP";
NETWORK
TITLE = da DB93.dbx52.0 a DB93.dbx52.7
      A     "MAP_DO".DB93_DBX052_0;
      =     "-387H1:LAMP";
      A     "MAP_DO".DB93_DBX052_1;
      =     "-387H2:LAMP";
      A     "MAP_DO".DB93_DBX052_2;
      =     #Temp1;
      A     "MAP_DO".DB93_DBX052_3;
      =     #Temp1;
      A     "MAP_DO".DB93_DBX052_4;
      =     "-363S4:LAMP";
      A     "MAP_DO".DB93_DBX052_5;
      =     #Temp1;
      A     "MAP_DO".DB93_DBX052_6;
      =     #Temp1;
      A     "MAP_DO".DB93_DBX052_7;
      =     #Temp1;
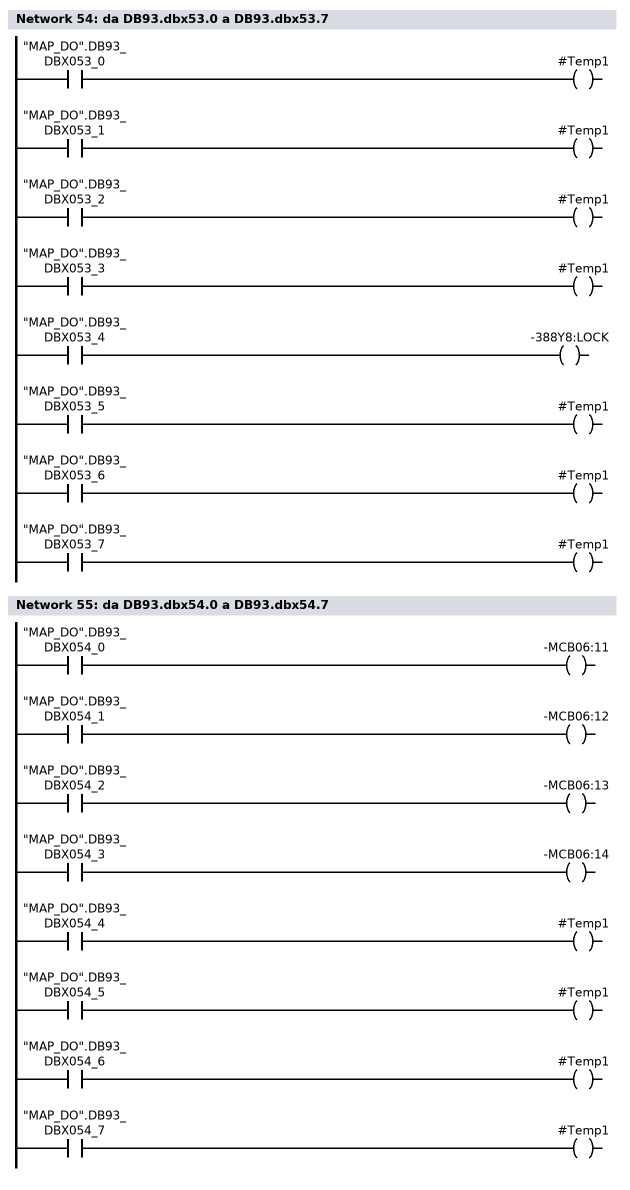
NETWORK
TITLE = da DB93.dbx53.0 a DB93.dbx53.7
      A     "MAP_DO".DB93_DBX053_0;
      =     #Temp1;
      A     "MAP_DO".DB93_DBX053_1;
      =     #Temp1;
      A     "MAP_DO".DB93_DBX053_2;
      =     #Temp1;
      A     "MAP_DO".DB93_DBX053_3;
      =     #Temp1;
      A     "MAP_DO".DB93_DBX053_4;
      =     "-388Y8:LOCK";
      A     "MAP_DO".DB93_DBX053_5;
      =     #Temp1;
      A     "MAP_DO".DB93_DBX053_6;
      =     #Temp1;
      A     "MAP_DO".DB93_DBX053_7;
      =     #Temp1;
NETWORK
TITLE = da DB93.dbx54.0 a DB93.dbx54.7
      A     "MAP_DO".DB93_DBX054_0;
      =     "-MCB06:11";
      A     "MAP_DO".DB93_DBX054_1;
      =     "-MCB06:12";
      A     "MAP_DO".DB93_DBX054_2;
      =     "-MCB06:13";
      A     "MAP_DO".DB93_DBX054_3;
      =     "-MCB06:14";
      A     "MAP_DO".DB93_DBX054_4;
      =     #Temp1;
      A     "MAP_DO".DB93_DBX054_5;
      =     #Temp1;
      A     "MAP_DO".DB93_DBX054_6;
      =     #Temp1;
      A     "MAP_DO".DB93_DBX054_7;
      =     #Temp1;
NETWORK
TITLE = da DB93.dbx55.0 a DB93.dbx55.7
      A     "MAP_DO".DB93_DBX055_0;
      CLR;
      =     "-388Y2";
      A     "MAP_DO".DB93_DBX055_1;
      CLR;
      =     "-388Y1";
      A     "MAP_DO".DB93_DBX055_2;
      =     #Temp1;
      A     "MAP_DO".DB93_DBX055_3;
      =     #Temp1;
      A     "MAP_DO".DB93_DBX055_4;
      =     #Temp1;
      A     "MAP_DO".DB93_DBX055_5;
      =     #Temp1;
      A     "MAP_DO".DB93_DBX055_6;
      =     #Temp1;
      A     "MAP_DO".DB93_DBX055_7;
      =     #Temp1;
NETWORK
TITLE = da DB93.dbx56.0 a DB93.dbx56.7
NETWORK
TITLE = da DB93.dbx57.0 a DB93.dbx57.7
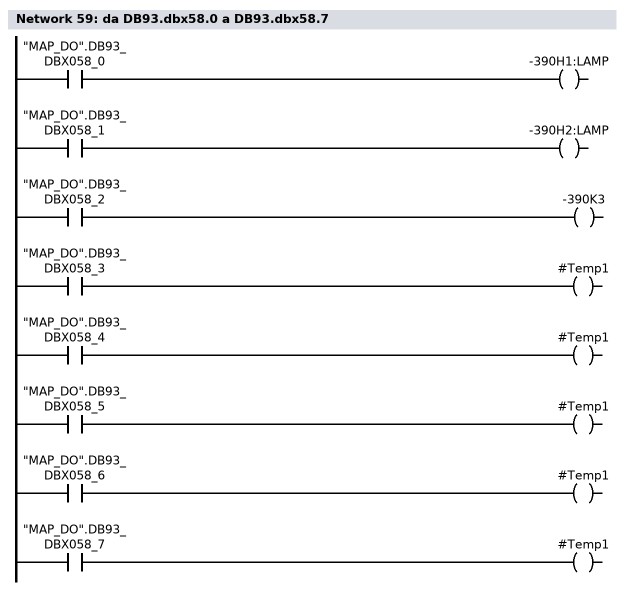
NETWORK
TITLE = da DB93.dbx58.0 a DB93.dbx58.7
      A     "MAP_DO".DB93_DBX058_0;
      =     "-390H1:LAMP";
      A     "MAP_DO".DB93_DBX058_1;
      =     "-390H2:LAMP";
      A     "MAP_DO".DB93_DBX058_2;
      =     "-390K3";
      A     "MAP_DO".DB93_DBX058_3;
      =     #Temp1;
      A     "MAP_DO".DB93_DBX058_4;
      =     #Temp1;
      A     "MAP_DO".DB93_DBX058_5;
      =     #Temp1;
      A     "MAP_DO".DB93_DBX058_6;
      =     #Temp1;
      A     "MAP_DO".DB93_DBX058_7;
      =     #Temp1;
NETWORK
TITLE = da DB93.dbx59.0 a DB93.dbx59.7
END_FUNCTION

FUNCTION "Increase-decrease" : VOID	// FC 100
TITLE = INCREASE - DECREASE FUNCTION
AUTHOR : Milesi
VERSION : 0.1
VAR_INPUT
  UP_LIMIT : REAL ;
  DOWN_LIMIT : REAL ;
END_VAR
VAR_IN_OUT
  INCREASE : BOOL ;
  DECREASE : BOOL ;
  CLOCK_FLAG : BOOL ;
  AUX_FLAG : BOOL ;
  OUT : REAL ;
END_VAR
BEGIN
NETWORK
TITLE = VALUE INCREASE
      AN    #INCREASE;
      JC    _001;
      A     #CLOCK_FLAG;
      FP    #AUX_FLAG;
      JCN   _001;
      L     #OUT;
      L     #UP_LIMIT;
      >=R;
      JC    _001;
      L     #OUT;
      L     1.000000e+00;
      +R;
      T     #OUT;
      JU    END;
_001: T     #OUT;
END:  NOP   0;
NETWORK
TITLE = VALUE DECREASE
      AN    #DECREASE;
      JC    _002;
      A     #CLOCK_FLAG;
      FP    #AUX_FLAG;
      JCN   _002;
      A(;
      L     #OUT;
      L     #DOWN_LIMIT;
      <=R;
      );
      JC    _002;
      L     #OUT;
      L     1.000000e+00;
      -R;
      T     #OUT;
      JU    END1;
_002: T     #OUT;
END1: NOP   0;
END_FUNCTION

FUNCTION "Flip-Flop" : VOID	// FC 101
TITLE = FLIP-FLOP FUNCTION
AUTHOR : Milesi
VERSION : 0.1
VAR_IN_OUT
  INPUT : BOOL ;
  MEM_FLAG1 : BOOL ;
  MEM_FLAG2 : BOOL ;
  OUTPUT : BOOL ;
END_VAR
BEGIN
NETWORK
TITLE = FLIP-FLOP
      A     #INPUT;
      AN    #MEM_FLAG1;
      S     #OUTPUT;
      AN    #INPUT;
      A     #OUTPUT;
      S     #MEM_FLAG2;
      A     #INPUT;
      A     #OUTPUT;
      A     #MEM_FLAG2;
      R     #OUTPUT;
      R     #MEM_FLAG2;
      S     #MEM_FLAG1;
      AN    #INPUT;
      A     #MEM_FLAG1;
      R     #MEM_FLAG1;
END_FUNCTION

FUNCTION "Ramp" : VOID	// FC 102
TITLE = RAMP FUNCTION
AUTHOR : Milesi
VERSION : 3.0
VAR_INPUT
  INPUT_10000 : REAL ;
  UP_DOWN_sec : REAL ;
  NORMAL_STOP_sec : REAL ;
  QUICK_STOP_sec : REAL ;
END_VAR
VAR_OUTPUT
  HOLD_LAMP : BOOL ;
  FIXED_RAMP : BOOL ;
END_VAR
VAR_IN_OUT
  RAMP_ENABLE : BOOL ;
  SLOW_DOWN : BOOL ;
  QUICK_STOP : BOOL ;
  HOLD : BOOL ;
  HOLD_FLAG : BOOL ;
  HOLD_FLAG_1 : BOOL ;
  OUTPUT_REAL_10000 : REAL ;
  OUTPUT_DINT_10000 : DINT ;
  OUTPUT_REAL_100 : REAL ;
  MEM_FLAG1 : BOOL ;
  MEM_FLAG2 : BOOL ;
  MEM_FLAG3 : BOOL ;
  MEM_FLAG4 : BOOL ;
  MEM_FLAG5 : BOOL ;
  MEM_FLAG6 : BOOL ;
END_VAR
VAR_TEMP
  UP_DOWN_STEP : REAL ;
  NORMAL_STOP_STEP : REAL ;
  QUICK_STOP_STEP : REAL ;
  DEADBAND_UP : REAL ;
  DEADBAND_DOWN : REAL ;
END_VAR
BEGIN
NETWORK
TITLE = RAMP INPUT VALUE
      L     #INPUT_10000;
      AN    #SLOW_DOWN;
      JC    BLO1;
      L     #INPUT_10000;
      L     2.000000e+00;
      /R;
BLO1: T     #INPUT_10000;
NETWORK
TITLE = RAMP UP STEP VALUE
      L     1.000000e+03;
      L     #UP_DOWN_sec;
      /R;
      T     #UP_DOWN_STEP;
NETWORK
TITLE = NORMAL RAMP DOWN STEP VALUE
      L     1.000000e+03;
      L     #NORMAL_STOP_sec;
      /R;
      T     #NORMAL_STOP_STEP;
NETWORK
TITLE = QUICK RAMP DOWN STEP VALUE
      L     1.000000e+03;
      L     #QUICK_STOP_sec;
      /R;
      T     #QUICK_STOP_STEP;
NETWORK
TITLE = RAMP HOLD
      CALL  "Flip-Flop" (
           INPUT                    := #HOLD_FLAG_1,
           MEM_FLAG1                := #MEM_FLAG1,
           MEM_FLAG2                := #MEM_FLAG2,
           OUTPUT                   := #HOLD_FLAG);
      NOP   0;
NETWORK
TITLE = RAMP HOLD LAMP
      A     #HOLD_FLAG;
      =     #HOLD_LAMP;
NETWORK
TITLE = RAMP HOLD RESET
      AN    #RAMP_ENABLE;
      A     #HOLD_FLAG;
      O;
      A     #RAMP_ENABLE;
      A     #HOLD;
      =     #HOLD_FLAG_1;
NETWORK
TITLE = FIXED RAMP CONTROL
      L     #INPUT_10000;
      L     1.000000e+02;
      +R;
      T     #DEADBAND_UP;
      L     #INPUT_10000;
      L     1.000000e+02;
      -R;
      T     #DEADBAND_DOWN;
      A(;
      A(;
      L     #OUTPUT_REAL_10000;
      L     #DEADBAND_UP;
      <=R;
      );
      A(;
      L     #OUTPUT_REAL_10000;
      L     #DEADBAND_DOWN;
      >=R;
      );
      O     #HOLD_FLAG;
      );
      AN    #SLOW_DOWN;
      =     #FIXED_RAMP;
NETWORK
TITLE = RAMP INCREASE - DECREASE
      A     #RAMP_ENABLE;
      AN    #HOLD_FLAG;
      JCN   END;
      L     #OUTPUT_REAL_10000;
      L     #INPUT_10000;
      <R;
      JC    UP;
      L     #OUTPUT_REAL_10000;
      L     #INPUT_10000;
      >R;
      JC    DOWN;
      JU    END;
UP:   A     "M1.0";
      FP    #MEM_FLAG3;
      JCN   END;
      L     #OUTPUT_REAL_10000;
      L     #UP_DOWN_STEP;
      +R;
      T     #OUTPUT_REAL_10000;
      JU    END;
DOWN: A     "M1.0";
      FP    #MEM_FLAG6;
      JCN   END;
      L     #OUTPUT_REAL_10000;
      L     #UP_DOWN_STEP;
      -R;
      T     #OUTPUT_REAL_10000;
END:  NOP   0;
NETWORK
TITLE = RAMP NORMAL STOP 
      A(;
      O     #RAMP_ENABLE;
      O     #QUICK_STOP;
      );
      JC    END1;
      A     "M1.0";
      FP    #MEM_FLAG5;
      JCN   END1;
      L     #OUTPUT_REAL_10000;
      L     #NORMAL_STOP_STEP;
      -R;
      T     #OUTPUT_REAL_10000;
      L     0.000000e+00;
      <=R;
      JCN   END1;
      L     0.000000e+00;
      T     #OUTPUT_REAL_10000;
END1: NOP   0;
NETWORK
TITLE = RAMP QUICK STOP
      A(;
      O     #RAMP_ENABLE;
      ON    #QUICK_STOP;
      );
      JC    END2;
      A     "M1.0";
      FP    #MEM_FLAG6;
      JCN   END2;
      L     #OUTPUT_REAL_10000;
      L     #QUICK_STOP_STEP;
      -R;
      T     #OUTPUT_REAL_10000;
      L     0.000000e+00;
      <=R;
      JCN   END2;
      L     0.000000e+00;
      T     #OUTPUT_REAL_10000;
END2: NOP   0;
NETWORK
TITLE = RAMP OUTPUT
      L     #OUTPUT_REAL_10000;
      RND;
      T     #OUTPUT_DINT_10000;
      L     #OUTPUT_REAL_10000;
      L     1.000000e+02;
      /R;
      T     #OUTPUT_REAL_100;
END_FUNCTION

FUNCTION "16 Bit Filter" : VOID	// FC 103
TITLE = 16 BIT FILTER FUNCTION
AUTHOR : Milesi
VERSION : 0.1
VAR_INPUT
  INPUT_VALUE : INT ;
  K_FILTER : INT ;
END_VAR
VAR_IN_OUT
  OUTPUT_VALUE : INT ;
  AUX_WORD1 : INT ;
  AUX_WORD2 : INT ;
END_VAR
BEGIN
NETWORK
TITLE = ADD VALUE
      L     #INPUT_VALUE;
      L     #AUX_WORD1;
      +I;
      T     #AUX_WORD1;
NETWORK
TITLE = COUNTER INCREASE
      L     #AUX_WORD2;
      L     1;
      +I;
      T     #AUX_WORD2;
      A(;
      L     #AUX_WORD2;
      L     #K_FILTER;
      >=I;
      );
      JCN   END;
NETWORK
TITLE = OUTPUT VALUE AND RESET
      L     #AUX_WORD1;
      L     #K_FILTER;
      /I;
      T     #OUTPUT_VALUE;
      L     0;
      T     #AUX_WORD1;
      T     #AUX_WORD2;
END:  NOP   0;
END_FUNCTION

FUNCTION "Diameter calculation" : VOID	// FC 105
TITLE = DIAMETER CALCULATION FUNCTION
AUTHOR : Milesi
VERSION : 3.0
VAR_INPUT
  Enable : BOOL ;
  Linear_Speed : REAL ;
  Bobbin_Speed : REAL ;
  Flange_Diameter : REAL ;
  Min_Diameter_Ratio : REAL ;
  K_Filter : REAL ;
END_VAR
VAR_IN_OUT
  Diameter_out : REAL ;
  Filter_Aux_1 : REAL ;
  Filter_Aux_2 : REAL ;
END_VAR
VAR_TEMP
  Diameter_Aux : REAL ;
  Min_Diameter : REAL ;
END_VAR
BEGIN
NETWORK
TITLE = DIAMETER CALCULATION
      AN    #Enable;
      JC    END;
      L     #Linear_Speed;
      L     #Bobbin_Speed;
      /R;
      L     3.141592e+00;
      *R;
      L     1.000000e+02;
      *R;
      T     #Diameter_Aux;
NETWORK
TITLE = LIMITS
      A(;
      L     #Flange_Diameter;
      L     #Min_Diameter_Ratio;
      /R;
      T     #Min_Diameter;
      );
      A(;
      L     #Diameter_Aux;
      L     #Min_Diameter;
      >=R;
      );
      JC    _001;
      L     #Min_Diameter;
      T     #Diameter_Aux;
_001: A(;
      L     #Diameter_Aux;
      L     #Flange_Diameter;
      <=R;
      );
      JC    _002;
      L     #Flange_Diameter;
      T     #Diameter_Aux;
_002: NOP   0;
NETWORK
TITLE = FILTER
      L     #Diameter_Aux;
      L     #Filter_Aux_1;
      +R;
      T     #Filter_Aux_1;
      L     #Filter_Aux_2;
      L     1.000000e+00;
      +R;
      T     #Filter_Aux_2;
      A(;
      L     #Filter_Aux_2;
      L     #K_Filter;
      >=R;
      );
      JCN   END1;
      L     #Filter_Aux_1;
      L     #K_Filter;
      /R;
      T     #Diameter_out;
      L     0.000000e+00;
      T     #Filter_Aux_1;
      T     #Filter_Aux_2;
END1: BEU;
END:  L     0.000000e+00;
      T     #Filter_Aux_1;
      T     #Filter_Aux_2;
END_FUNCTION

FUNCTION "Increase-decrease head" : VOID	// FC 106
TITLE = INCREASE - DECREASE HEAD FUNCTION
AUTHOR : Milesi
VERSION : 0.1
VAR_INPUT
  UP_LIMIT : REAL ;
  DOWN_LIMIT : REAL ;
  HEAD_MAX_RPM : REAL ;
END_VAR
VAR_IN_OUT
  INCREASE : BOOL ;
  DECREASE : BOOL ;
  CLOCK_FLAG : BOOL ;
  AUX_FLAG : BOOL ;
  HEAD_REAL_RPM : REAL ;
  OUT : REAL ;
END_VAR
BEGIN
NETWORK
TITLE = VALUE INCREASE
      AN    #INCREASE;
      JC    END;
      A     #CLOCK_FLAG;
      FP    #AUX_FLAG;
      JCN   END;
      L     #OUT;
      L     #UP_LIMIT;
      >=R;
      JC    END;
      L     #OUT;
      L     1.000000e+00;
      +R;
      T     #OUT;
END:  NOP   0;
NETWORK
TITLE = VALUE DECREASE
      A(;
      L     #HEAD_REAL_RPM;
      L     #HEAD_MAX_RPM;
      >=R;
      );
      ON    #DECREASE;
      JC    END1;
      A     #CLOCK_FLAG;
      FP    #AUX_FLAG;
      JCN   END1;
      A(;
      L     #OUT;
      L     #DOWN_LIMIT;
      <=R;
      );
      JC    END1;
      L     #OUT;
      L     1.000000e+00;
      -R;
      T     #OUT;
END1: NOP   0;
END_FUNCTION

FUNCTION "32 Bit filter" : VOID	// FC 108
TITLE = 32 BIT FILTER  FUNCTION
AUTHOR : Milesi
VERSION : 0.1
VAR_INPUT
  INPUT_VALUE : REAL ;
  K_FILTER : REAL ;
END_VAR
VAR_IN_OUT
  OUTPUT_VALUE : REAL ;
  AUX_TOTAL_REAL : REAL ;
  AUX_COUNT : REAL ;
END_VAR
BEGIN
NETWORK
TITLE = ADD VALUE
      L     #INPUT_VALUE;
      L     #AUX_TOTAL_REAL;
      +R;
      T     #AUX_TOTAL_REAL;
NETWORK
TITLE = COUNTER INCREASE
      L     #AUX_COUNT;
      L     1.000000e+00;
      +R;
      T     #AUX_COUNT;
      A(;
      L     #AUX_COUNT;
      L     #K_FILTER;
      >=R;
      );
      JCN   END;
NETWORK
TITLE = OUTPUT VALUE AND RESET
      L     #AUX_TOTAL_REAL;
      L     #K_FILTER;
      /R;
      T     #OUTPUT_VALUE;
      L     0.000000e+00;
      T     #AUX_TOTAL_REAL;
      T     #AUX_COUNT;
END:  NOP   0;
END_FUNCTION

FUNCTION "Capstan linear speed" : VOID	// FC 112
TITLE = CAPSTAN LINEAR SPEED CALCULATION FUNCTION
AUTHOR : Milesi
VERSION : 0.1
VAR_INPUT
  Enable : BOOL ;
  Capstan_pulley_diameter : REAL ;
  Cable_diameter : REAL ;
  Input_speed : REAL ;
  Input_speed_resolution : REAL ;
  Max_line_speed : REAL ;
  K_filter : REAL ;
END_VAR
VAR_IN_OUT
  Added_value : REAL ;
  Counter_increase : REAL ;
  Filtered_linear_speed : REAL ;
END_VAR
VAR_TEMP
  Cable_diameter_const : REAL ;
  Actual_linear_speed : REAL ;
END_VAR
BEGIN
NETWORK
TITLE = CABLE DIAMETER CONSTANT
//             Capstan pulley Ш + Cable Ш
//K (Cable Ш)= --------------------------
//                 Capstan pulley Ш
      AN    #Enable;
      JC    _001;
      L     #Capstan_pulley_diameter;
      L     #Cable_diameter;
      +R;
      L     #Capstan_pulley_diameter;
      /R;
      T     #Cable_diameter_const;
NETWORK
TITLE = LINEAR SPEED CALCULATION
//                             Input_speed               
//Linear Speed (mt/min) = ----------------------   * Max_line_speed * K (Cable Ш)
//                        Input_speed_resolution        
      L     #Input_speed;
      L     #Input_speed_resolution;
      /R;
      L     #Max_line_speed;
      *R;
      L     #Cable_diameter_const;
      *R;
      JU    END;
_001: L     0.000000e+00;
END:  T     #Actual_linear_speed;
NETWORK
TITLE = FILTER + OUTPUT VALUE
      L     #Actual_linear_speed;
      L     #Added_value;
      +R;
      T     #Added_value;
      L     #Counter_increase;
      L     1.000000e+00;
      +R;
      T     #Counter_increase;
      A(;
      L     #Counter_increase;
      L     #K_filter;
      >=R;
      );
      JCN   END1;
      L     #Added_value;
      L     #K_filter;
      /R;
      T     #Filtered_linear_speed;
      L     0.000000e+00;
      T     #Added_value;
      T     #Counter_increase;
END1: NOP   0;
END_FUNCTION

FUNCTION "Bobbins wire management" : VOID	// FC 113
TITLE = BOBBIN WIRE MANAGEMENT FUNCTION
AUTHOR : Milesi
VERSION : 0.1
VAR_INPUT
  Enable : BOOL ;	//Enable function
  EnableWireBreakAlm : BOOL ;	//Enable no rotation alarm detecting
  Pulse : BOOL ;	//Input for rotation sensor
  ResetAlarm : BOOL ;	//Acknoledge and reset of no rotation alarm
  DelayTime : S5TIME ;	//Delay alarm before no rotation alarm
  StorageTimer : TIMER ;	//Timer for no rotation alarm
END_VAR
VAR_IN_OUT
  NumMovingBobbins : INT ;	//Register for number total of bobbins running
  EnableCountBobbins : BOOL ;	//Start of counter of total bobbins running (0=start counter; 1=bobbin detected)
  Mem : BOOL ;	//Aux Memory for rise up and fall down signal generation
  BobbinMoving : BOOL ;	//Bobbin moving detected
  ALARM : BOOL ;	//Bobbin no rotation alarm
END_VAR
VAR_TEMP
  Pulse_int : BOOL ;	//Pulse front
END_VAR
BEGIN
NETWORK
TITLE = Rise up and Fall down of pulse caching
      A     #Pulse;
      AN    #Mem;
      O;
      AN    #Pulse;
      A     #Mem;
      =     #Pulse_int;
NETWORK
TITLE = Bobbin moving
      A     #Pulse_int;
      S     #BobbinMoving;
      A(;
      ON    #Enable;
      O     #ALARM;
      );
      R     #BobbinMoving;
      NOP   0;
NETWORK
TITLE = No rotation alarm calculation
      A(;
      AN    #ResetAlarm;
      A     #Enable;
      A     #EnableWireBreakAlm;
      AN    #Pulse_int;
      L     #DelayTime;
      SD    #StorageTimer;
      NOP   0;
      NOP   0;
      NOP   0;
      A     #StorageTimer;
      );
      A     #BobbinMoving;
      S     #ALARM;
      A     #ResetAlarm;
      R     #ALARM;
      NOP   0;
NETWORK
TITLE = Pulse auxiliar memory
      A     #Pulse;
      =     #Mem;
NETWORK
TITLE = Number of moving Bobbins calculation
      A(;
      AN    #EnableCountBobbins;
      A     #BobbinMoving;
      JNB   _001;
      L     1;
      L     #NumMovingBobbins;
      +I;
      T     #NumMovingBobbins;
      AN    OV;
      SAVE;
      CLR;
_001: A     BR;
      );
      S     #EnableCountBobbins;
      AN    #Enable;
      R     #EnableCountBobbins;
      NOP   0;
END_FUNCTION

FUNCTION "Bobbin diameter calculat" : VOID	// FC 114
TITLE = BOBBIN DIAMETER CALCULATION FUNCTION
AUTHOR : Milesi
VERSION : 0.1
VAR_INPUT
  Enable : BOOL ;
  Pulse : BOOL ;
  Pulse_1minute : BOOL ;
  Reset : BOOL ;
  LinearSpeed : REAL ;
  CompattingFactorHMI : REAL ;
  MinDiameterLimit : REAL ;
  MaxDiameterLimit : REAL ;
  Pulses_number : INT ;
END_VAR
VAR_IN_OUT
  Mem : BOOL ;
  ImpulseForMinRegister : INT ;
  Diameter : INT ;
END_VAR
VAR_TEMP
  Cage_math_auxiliary : REAL ;
  Cable_compatting_costant : REAL ;
  Linear_Speed_Compatted : REAL ;
  Bobbin_rpm : REAL ;
  PulseXMin_Real : REAL ;
  PulsesNumber_Real : REAL ;
  Diameter_Real : REAL ;
  Pulse_imp : BOOL ;
END_VAR
BEGIN
NETWORK
TITLE = CABLE COMPACTING CONSTANT CALCULATION
//Linear speed read and adjusted by the compacting percentage is the following:
//
//                           LinearSpeedRead * CompactingPercent * 3mt/min  
//VelAdj = LinearSpeedRead -  ---------------------------------------------
//                                     100 * MaxLinearSpeed
//
//                            CompactingPercent * 3
//K Compacting Factor = (1 - ---------------------- )
//                            100 * MaxLinearSpeed 
//
//
//3mt/min is the "quantity" of influence determined by the compacting percentage 
//(0 - 3 mt/min : 0 - 100%)
//The max linear speed of this machine is 60 mt/min
//Then the K Compacting Factor can be reduced to :
//
//                           CompactingPercent
//K Compacting Factor = (1 - --------------- )
//                                 2000 
      L     #CompattingFactorHMI;
      L     2.000000e+03;
      /R;
      T     #Cage_math_auxiliary;
      L     1.000000e+00;
      L     #Cage_math_auxiliary;
      -R;
      T     #Cable_compatting_costant;
NETWORK
TITLE = ADJUSTED LINEAR SPEED CALCULATION
      L     #LinearSpeed;
      L     #Cable_compatting_costant;
      *R;
      T     #Linear_Speed_Compatted;
NETWORK
TITLE =
      A     #Enable;
      A     #Pulse;
      AN    #Mem;
      =     #Pulse_imp;
NETWORK
TITLE = BOBBIN DIAMETER CALCULATION
      AN    #Enable;
      JC    M107;
      A     #Pulse_1minute;
      JC    M006;
      A     #Pulse_imp;
      JNB   M007;
      L     #ImpulseForMinRegister;
      L     1;
      +I;
      T     #ImpulseForMinRegister;
      JU    M007;
M006: L     #ImpulseForMinRegister;
      ITD;
      DTR;
      T     #PulseXMin_Real;
      L     #Pulses_number;
      ITD;
      DTR;
      T     #PulsesNumber_Real;
      L     #PulseXMin_Real;
      L     #PulsesNumber_Real;
      /R;
      T     #Bobbin_rpm;
      L     #Linear_Speed_Compatted;
      L     #Bobbin_rpm;
      /R;
      L     1.000000e+03;
      *R;
      L     3.140000e+00;
      /R;
      T     #Diameter_Real;
      RND;
      T     #Diameter;
M107: L     0;
      T     #ImpulseForMinRegister;
M007: NOP   0;
NETWORK
TITLE = BOBBIN MINIMUM DIAMETER LIMIT 
      A(;
      L     #Diameter;
      L     #MinDiameterLimit;
      RND;
      <I;
      );
      JNB   _001;
      L     #MinDiameterLimit;
      RND;
      T     #Diameter;
_001: NOP   0;
NETWORK
TITLE = BOBBIN MAX DIAMETER LIMIT 
      A(;
      L     #Diameter;
      L     #MaxDiameterLimit;
      RND;
      >I;
      );
      JNB   _002;
      L     #MaxDiameterLimit;
      RND;
      T     #Diameter;
_002: NOP   0;
NETWORK
TITLE = BOBBIN DIAMETER RESET
      AN    #Reset;
      JC    _018;
      L     #MaxDiameterLimit;
      RND;
      T     #Diameter;
      L     0;
      T     #ImpulseForMinRegister;
_018: NOP   0;
NETWORK
TITLE =
      A     #Enable;
      A     #Pulse;
      S     #Mem;
      A     #Enable;
      AN    #Pulse;
      R     #Mem;
      NOP   0;
END_FUNCTION

FUNCTION "Motor status HMI" : VOID	// FC 115
TITLE = MOTOR STATUS CHECKING FOR HMI ANIMATION FUNCTION
AUTHOR : Milesi
VERSION : 0.1
VAR_INPUT
  Start : BOOL ;
  Fault : BOOL ;
END_VAR
VAR_IN_OUT
  Status_Reg : BYTE ;
END_VAR
VAR_TEMP
  temp : BOOL ;
END_VAR
BEGIN
NETWORK
TITLE =
      A     #Start;
      AN    #Fault;
      JNB   _001;
      L     1;
      T     #Status_Reg;
_001: NOP   0;
NETWORK
TITLE =
      A     #Fault;
      JNB   _002;
      L     2;
      T     #Status_Reg;
_002: NOP   0;
NETWORK
TITLE =
      AN    #Start;
      AN    #Fault;
      JNB   _003;
      L     0;
      T     #Status_Reg;
_003: NOP   0;
END_FUNCTION

FUNCTION "Rotation control" : VOID	// FC 200
TITLE = ROTATION CONTROL FUNCTION
AUTHOR : Milesi
VERSION : 0.1
VAR_INPUT
  Enable : BOOL ;
  Pulse : BOOL ;
  Reset : BOOL ;
  DelayTime : S5TIME ;
  StorageTimer : TIMER ;
END_VAR
VAR_IN_OUT
  Mem : BOOL ;
  ALARM : BOOL ;
END_VAR
VAR_TEMP
  Pulse_int : BOOL ;
END_VAR
BEGIN
NETWORK
TITLE =
      A     #Enable;
      A     #Pulse;
      AN    #Mem;
      O;
      A     #Enable;
      AN    #Pulse;
      A     #Mem;
      =     #Pulse_int;
NETWORK
TITLE =
      A(;
      A     #Enable;
      AN    #Pulse_int;
      L     #DelayTime;
      SS    #StorageTimer;
      AN    #Enable;
      R     #StorageTimer;
      NOP   0;
      NOP   0;
      A     #StorageTimer;
      );
      S     #ALARM;
      A     #Reset;
      R     #ALARM;
      NOP   0;
NETWORK
TITLE =
      A     #Enable;
      A     #Pulse;
      =     #Mem;
END_FUNCTION

